(* IEC 61131-3 sources: std_i2980_v2.06_cp053/Source/IMM/ieccontrol/HostCommunication, 9 files *)

(* ---- ABDataSet.pu ---- *)
IMPORT_OVER_LISTFILE
 GET_SYNC_REFTO
, ASSERT
, STOP_PROCESS_ALGORITHM
, cDataSetErr_NoAvailable
, cDataSetErr_NotAllowed
, cModeAutomatic
, cCompOperationMode
, tevLockUnlock
, tsHostHmi
, tsHostDataSet
, tnDataState
, tnOperationMode
, KSYS_Status
, FBLockUnlock

END_IMPORT

ALGORITHM_BLOCK ABDataSet #DUMMY_EDIT_BLOCK

SYSTEM_VAR
 sv_bInitDone : BOOL (* IEC initialisation is finished (after movement registration) *);
 sv_HostHmi : tsHostHmi;
 sv_DataSet : tsHostDataSet;
 sv_DataState : tnDataState (* State of machine / mold data read *);
 sv_OperationMode : tnOperationMode;
END_VAR

SYSTEM_OBJECT
 TaskVis : TASK;
 evLockUnlock : tevLockUnlock;
 erAssert : ALARM;
END_OBJECT

VAR
 mpbAllowMoldLoad : REFTO BOOL;
 mpbAllowMoldSave : REFTO BOOL;
 mpbAllowMachineLoad : REFTO BOOL;
 mpbAllowMachineSave : REFTO BOOL;
 mpbAllowSeqLoad : REFTO BOOL;
 mpbAllowSeqSave : REFTO BOOL;
 mbOpModeLockAvailable : BOOL;
 mDataActionsEnableAvailable : BOOL;
END_VAR

FUNCTION fIsOpModeAutoAllowed : BOOL
 #DUMMY_EDIT_BLOCK
#BEGIN_EDIT_BLOCK

fIsOpModeAutoAllowed := NOT (sv_DataSet.iCommand = cDataSetCmdLoadMold) OR (sv_DataSet.iCommand = cDataSetCmdLoadMachine);

;#END_EDIT_BLOCK END_FUNCTION

FUNCTION fCheckConditions : BOOL
 #DUMMY_EDIT_BLOCK
#BEGIN_EDIT_BLOCK
IF (sv_DataState <> nReady) THEN
    RETURN;
END_IF;

IF (NOT fIsOpModeAutoAllowed()) THEN
    IF (sv_OperationMode >= nHalfAutomatic) THEN
        RETURN;
    END_IF;
END_IF;

fCheckConditions := TRUE;

;#END_EDIT_BLOCK END_FUNCTION

FUNCTION fDisableAll : BOOL
 #DUMMY_EDIT_BLOCK

VAR_INPUT
 bDisable : BOOL;
END_VAR
#BEGIN_EDIT_BLOCK
IF (mDataActionsEnableAvailable) THEN
   mpbAllowMoldLoad^ := NOT bDisable;
   mpbAllowMoldSave^ := NOT bDisable;
   mpbAllowMachineLoad^ := NOT bDisable;
   mpbAllowMachineSave^ := NOT bDisable;
   mpbAllowSeqLoad^ := NOT bDisable;
   mpbAllowSeqSave^ := NOT bDisable;
END_IF;

;#END_EDIT_BLOCK END_FUNCTION

POSTUPDATE_ALGORITHM pInit ON TaskVis(1) WITH sv_HostHmi.dataSet.bAvailable

VAR
 b : BOOL;
 s : KSYS_Status;
 dummy : DINT;
 dummyRef : REFTO UDINT;
END_VAR
#BEGIN_EDIT_BLOCK
mDataActionsEnableAvailable := TRUE;
mpbAllowMoldLoad := GET_SYNC_REFTO("system.sv_DataActionsEnable.bMoldDataLoad", T#0s, s);
mDataActionsEnableAvailable := mDataActionsEnableAvailable AND (s = KSYS_Status_OK);
mpbAllowMoldSave := GET_SYNC_REFTO("system.sv_DataActionsEnable.bMoldDataSave", T#0s, s);
mDataActionsEnableAvailable := mDataActionsEnableAvailable AND (s = KSYS_Status_OK);
mpbAllowMachineLoad := GET_SYNC_REFTO("system.sv_DataActionsEnable.bMachineDataLoad", T#0s, s);
mDataActionsEnableAvailable := mDataActionsEnableAvailable AND (s = KSYS_Status_OK);
mpbAllowMachineSave := GET_SYNC_REFTO("system.sv_DataActionsEnable.bMachineDataSave", T#0s, s);
mDataActionsEnableAvailable := mDataActionsEnableAvailable AND (s = KSYS_Status_OK);
mpbAllowSeqLoad := GET_SYNC_REFTO("system.sv_DataActionsEnable.bSequenceDataLoad", T#0s, s);
mDataActionsEnableAvailable := mDataActionsEnableAvailable AND (s = KSYS_Status_OK);
mpbAllowSeqSave := GET_SYNC_REFTO("system.sv_DataActionsEnable.bSequenceDataSave", T#0s, s);
mDataActionsEnableAvailable := mDataActionsEnableAvailable AND (s = KSYS_Status_OK);

dummyRef := GET_SYNC_REFTO("system.sv_LockOperationModeAuto.sResourceLock.iLocked", T#0s, s);
mbOpModeLockAvailable := s = KSYS_Status_OK;

IF (evLockUnlock = EMPTY) THEN
   dummy := Print("HostCommunication.ABDataSet: binary incompatible! recompile FU with correct iecproject!");
   b := ASSERT(FALSE, erAssert);
END_IF;

;#END_EDIT_BLOCK END_ALGORITHM

POSTUPDATE_ALGORITHM pTrigger ON TaskVis(2) WITH sv_DataSet.iTrigger

VAR
 b : BOOL;
END_VAR
#BEGIN_EDIT_BLOCK
IF (sv_DataSet.iTrigger MOD 2 = 0) THEN
    RETURN;
END_IF;

sv_DataSet.iError := 0;
IF (NOT sv_bInitDone) THEN
    sv_DataSet.iError := cDataSetErr_NotAllowed;
ELSIF (NOT sv_HostHmi.dataSet.bAvailable) THEN
    sv_DataSet.iError := cDataSetErr_NoAvailable;
ELSIF ((sv_DataSet.iCommand < cDataSetCmdLoadMold) OR (sv_DataSet.iCommand > cDataSetCmdSaveMachine)) THEN
    sv_DataSet.iError := cDataSetErr_InvalidCommand;
ELSIF (NOT fCheckConditions()) THEN
    sv_DataSet.iError := cDataSetErr_NotAllowed;
END_IF;

IF (sv_DataSet.iError > 0) THEN
    sv_DataSet.iTrigger := sv_DataSet.iTrigger + 1;
    RETURN;
END_IF;

b := fDisableAll(TRUE);

START_PROCESS_ALGORITHM(paRun);

;#END_EDIT_BLOCK END_ALGORITHM

PROCESS_ALGORITHM paRun ON TaskVis

VAR
 iStep : DINT;
 cnt : DINT;
 fbLockUnlock : FBLockUnlock;
 b : BOOL;
END_VAR
#BEGIN_EDIT_BLOCK
IF (iStep = 0) THEN
    IF (mbOpModeLockAvailable) THEN
        // op-mode will be locked by HMI (CR_0074160)
        iStep := 20;
    ELSE
        IF (NOT fIsOpModeAutoAllowed()) THEN
           fbLockUnlock.DeviceId.CompId := cCompOperationMode;
           fbLockUnlock.DeviceId.IndexId := 1;
           fbLockUnlock.MoveDir := cModeAutomatic;
           fbLockUnlock.MoveId := cModeAutomatic;
           fbLockUnlock(Mode := nLockAbort);
        END_IF;
        cnt := 10;
        iStep := 10;
    END_IF;
END_IF;

// CR_0074160: actually it is not possible to ensure there is no other load- or save-action in progress
// as a workaround lock the recipemask buttons and wait a second, then check conditions again
IF (iStep = 10) THEN
    cnt := cnt - 1;
    IF (cnt = 0) THEN
        iStep := 20;
    END_IF;
END_IF;

IF (iStep = 20) THEN
    IF (NOT fCheckConditions()) THEN
        sv_DataSet.iError := cDataSetErr_NotAllowed;
        iStep := 1000;
    ELSE
        iStep := 30;
    END_IF;
END_IF;

IF (iStep = 30) THEN
    sv_HostHmi.dataSet.iCommand := sv_DataSet.iCommand;
    sv_HostHmi.dataSet.sFile := sv_DataSet.sFile;
    sv_HostHmi.dataSet.iTrigger := sv_HostHmi.dataSet.iTrigger + 1;
    iStep := 40;
END_IF;

IF (iStep = 40) THEN
    IF (sv_HostHmi.dataSet.iTrigger MOD 2 = 0) THEN
        sv_DataSet.iError := sv_HostHmi.dataSet.iError;
        iStep := 1000;
    END_IF;
END_IF;

IF (iStep = 1000) THEN
    b := fDisableAll(FALSE);
    IF (NOT mbOpModeLockAvailable) THEN
        fbLockUnlock(Mode := nUnlock);
    END_IF;
    sv_DataSet.iTrigger := sv_DataSet.iTrigger + 1;
    iStep := 0;
    STOP_PROCESS_ALGORITHM();
END_IF;

;#END_EDIT_BLOCK END_ALGORITHM

END_ALGORITHM_BLOCK

#END_OF_IEC_PART

@Puma @IecEditor 6 159 @Pou 25
@@@BEG_Comment@@@

@@@END_Comment@@@

@BEG_Contents

@BEG_Func
@RT(17)FuncTreeContainer
3
@Var @RT(14)GET_SYNC_REFTO @RT(0) @T @T @DERIVED 0 @F @RT(22)KEBA_STANDARD_FUNCTION @F
@T
@BEG_Attrib
0 @RT(0) @RT(0)
@END_Attrib
1 1 @F @F @F @F

@Var @RT(6)ASSERT @RT(0) @T @T @DERIVED 0 @F @RT(8)FUNCTION @F
@T
@BEG_Attrib
0 @RT(0) @RT(0)
@END_Attrib
1 1 @F @F @F @F

@Var @RT(22)STOP_PROCESS_ALGORITHM @RT(0) @T @T @DERIVED 0 @F @RT(23)KEBA_STANDARD_PROCEDURE @F
@T
@BEG_Attrib
0 @RT(0) @RT(0)
@END_Attrib
1 1 @F @F @F @F

@END_Func

@BEG_Const
@RT(18)ConstTreeContainer
4
@Var @RT(23)cDataSetErr_NoAvailable @RT(0) @T @F @DT @RT(4)DINT @RT(0) @T @T @BASIC 0 @F
@F @F
@T
@BEG_Attrib
0 @RT(1)1 @RT(0)
@END_Attrib
1 1 @F @F @F @F

@Var @RT(22)cDataSetErr_NotAllowed @RT(0) @T @F @DT @RT(4)DINT @RT(0) @T @T @BASIC 0 @F
@F @F
@T
@BEG_Attrib
0 @RT(1)3 @RT(0)
@END_Attrib
1 1 @F @F @F @F

@Var @RT(14)cModeAutomatic @RT(0) @T @F @DT @RT(4)DINT @RT(0) @T @T @BASIC 0 @F
@F @F
@T
@BEG_Attrib
0 @RT(2)23 @RT(50)for locking/unlocking half and full automatic mode
@END_Attrib
1 1 @F @F @F @F

@Var @RT(18)cCompOperationMode @RT(0) @T @F @DT @RT(4)DINT @RT(0) @T @T @BASIC 0 @F
@F @F
@T
@BEG_Attrib
0 @RT(3)111 @RT(24)Component Operation Mode
@END_Attrib
1 1 @F @F @F @F

@END_Const

@BEG_Export

@BEG_Kind
@ALGORITHM_BLOCK @RT(9)ABDataSet @STRUCTURED_TEXT
@RT(0) @RT(0) @RT(0)
@END_Kind

@BEG_Dcl
@RT(16)DclTreeContainer
16
@Var @RT(7)TaskVis @RT(0) @T @T @RENAMED 0 @T @T @DT @RT(4)TASK @RT(0) @T @T @BASIC 0 @F
@F @F
@T
@BEG_Attrib
3 @RT(0) @RT(0) @RT(0)
@END_Attrib
1 7 @F @F @F @F

@Var @RT(12)sv_bInitDone @RT(0) @T @F @DT @RT(4)BOOL @RT(0) @T @T @BASIC 0 @F
@F @F
@T
@BEG_Attrib
3 @RT(0) @RT(60)IEC initialisation is finished (after movement registration) @RT(0)
@END_Attrib
1 8 @F @F @F @F

@Var @RT(12)evLockUnlock @RT(0) @T @T @DERIVED 0 @T @T @DT @RT(13)tevLockUnlock @RT(0) @T @T @UNKNOWN 0 @F
@F @F
@T
@BEG_Attrib
3 @RT(0) @RT(0) @RT(0)
@END_Attrib
1 7 @F @F @F @F

@Var @RT(10)sv_HostHmi @RT(0) @T @T @DERIVED 0 @T @T @DT @RT(9)tsHostHmi @RT(0) @T @T @UNKNOWN 0 @F
@F @F
@T
@BEG_Attrib
3 @RT(0) @RT(0) @RT(0)
@END_Attrib
1 8 @F @F @F @F

@Var @RT(10)sv_DataSet @RT(0) @T @T @DERIVED 0 @T @T @DT @RT(13)tsHostDataSet @RT(0) @T @T @UNKNOWN 0 @F
@F @F
@T
@BEG_Attrib
3 @RT(0) @RT(0) @RT(0)
@END_Attrib
1 8 @F @F @F @F

@Var @RT(12)sv_DataState @RT(0) @T @T @DERIVED 0 @T @T @DT @RT(11)tnDataState @RT(0) @T @T @UNKNOWN 0 @F
@F @F
@T
@BEG_Attrib
3 @RT(0) @RT(33)State of machine / mold data read @RT(0)
@END_Attrib
1 8 @F @F @F @F

@Var @RT(16)sv_OperationMode @RT(0) @T @T @DERIVED 0 @T @T @DT @RT(15)tnOperationMode @RT(0) @T @T @UNKNOWN 0 @F
@F @F
@T
@BEG_Attrib
3 @RT(0) @RT(0) @RT(0)
@END_Attrib
1 8 @F @F @F @F

@Var @RT(8)erAssert @RT(0) @T @F @DT @RT(5)ALARM @RT(0) @T @T @BASIC 0 @F
@F @F
@T
@BEG_Attrib
3 @RT(0) @RT(0) @RT(0)
@END_Attrib
1 7 @F @F @F @F

@Var @RT(16)mpbAllowMoldLoad @RT(0) @T @T @REFTO 0 @T @DT @RT(4)BOOL @RT(0) @T @T @BASIC 0 @F
@F @F
@T
@BEG_Attrib
3 @RT(0) @RT(0) @RT(0)
@END_Attrib
1 0 @F @F @F @F

@Var @RT(16)mpbAllowMoldSave @RT(0) @T @T @REFTO 0 @T @DT @RT(4)BOOL @RT(0) @T @T @BASIC 0 @F
@F @F
@T
@BEG_Attrib
3 @RT(0) @RT(0) @RT(0)
@END_Attrib
1 0 @F @F @F @F

@Var @RT(19)mpbAllowMachineLoad @RT(0) @T @T @REFTO 0 @T @DT @RT(4)BOOL @RT(0) @T @T @BASIC 0 @F
@F @F
@T
@BEG_Attrib
3 @RT(0) @RT(0) @RT(0)
@END_Attrib
1 0 @F @F @F @F

@Var @RT(19)mpbAllowMachineSave @RT(0) @T @T @REFTO 0 @T @DT @RT(4)BOOL @RT(0) @T @T @BASIC 0 @F
@F @F
@T
@BEG_Attrib
3 @RT(0) @RT(0) @RT(0)
@END_Attrib
1 0 @F @F @F @F

@Var @RT(15)mpbAllowSeqLoad @RT(0) @T @T @REFTO 0 @T @DT @RT(4)BOOL @RT(0) @T @T @BASIC 0 @F
@F @F
@T
@BEG_Attrib
3 @RT(0) @RT(0) @RT(0)
@END_Attrib
1 0 @F @F @F @F

@Var @RT(15)mpbAllowSeqSave @RT(0) @T @T @REFTO 0 @T @DT @RT(4)BOOL @RT(0) @T @T @BASIC 0 @F
@F @F
@T
@BEG_Attrib
3 @RT(0) @RT(0) @RT(0)
@END_Attrib
1 0 @F @F @F @F

@Var @RT(21)mbOpModeLockAvailable @RT(0) @T @F @DT @RT(4)BOOL @RT(0) @T @T @BASIC 0 @F
@F @F
@T
@BEG_Attrib
3 @RT(0) @RT(0) @RT(0)
@END_Attrib
1 0 @F @F @F @F

@Var @RT(27)mDataActionsEnableAvailable @RT(0) @T @F @DT @RT(4)BOOL @RT(0) @T @T @BASIC 0 @F
@F @F
@T
@BEG_Attrib
3 @RT(0) @RT(0) @RT(0)
@END_Attrib
1 0 @F @F @F @F

@END_Dcl

@END_Export

@BEG_Body

6

@BEG_Export

@BEG_Algo
@FUNCTION @RT(20)fIsOpModeAutoAllowed @STRUCTURED_TEXT
@RT(4)BOOL @RT(0) @RT(0) @F @F
@END_Algo

@BEG_Dcl
@RT(16)DclTreeContainer
0
@END_Dcl

@END_Export

@BEG_Export

@BEG_Algo
@FUNCTION @RT(16)fCheckConditions @STRUCTURED_TEXT
@RT(4)BOOL @RT(0) @RT(0) @F @F
@END_Algo

@BEG_Dcl
@RT(16)DclTreeContainer
0
@END_Dcl

@END_Export

@BEG_Export

@BEG_Algo
@FUNCTION @RT(11)fDisableAll @STRUCTURED_TEXT
@RT(4)BOOL @RT(0) @RT(0) @F @F
@END_Algo

@BEG_Dcl
@RT(16)DclTreeContainer
1
@Var @RT(8)bDisable @RT(0) @T @F @DT @RT(4)BOOL @RT(0) @T @T @BASIC 0 @F
@F @F
@T
@BEG_Attrib
3 @RT(0) @RT(0) @RT(0)
@END_Attrib
1 1 @F @F @F @F

@END_Dcl

@END_Export

@BEG_Export

@BEG_Algo
@POSTUPDATE_ALGORITHM @RT(5)pInit @STRUCTURED_TEXT
@RT(0) @RT(29)sv_HostHmi.dataSet.bAvailable @RT(10)TaskVis(1) @F @F
@END_Algo

@BEG_Dcl
@RT(16)DclTreeContainer
4
@Var @RT(1)b @RT(0) @T @F @DT @RT(4)BOOL @RT(0) @T @T @BASIC 0 @F
@F @F
@T
@BEG_Attrib
3 @RT(0) @RT(0) @RT(0)
@END_Attrib
1 0 @F @F @F @F

@Var @RT(1)s @RT(0) @T @T @DERIVED 0 @T @T @DT @RT(11)KSYS_Status @RT(0) @T @T @UNKNOWN 0 @F
@F @F
@T
@BEG_Attrib
3 @RT(0) @RT(0) @RT(0)
@END_Attrib
1 0 @F @F @F @F

@Var @RT(5)dummy @RT(0) @T @F @DT @RT(4)DINT @RT(0) @T @T @BASIC 0 @F
@F @F
@T
@BEG_Attrib
3 @RT(0) @RT(0) @RT(0)
@END_Attrib
1 0 @F @F @F @F

@Var @RT(8)dummyRef @RT(0) @T @T @REFTO 0 @T @DT @RT(5)UDINT @RT(0) @T @T @BASIC 0 @F
@F @F
@T
@BEG_Attrib
3 @RT(0) @RT(0) @RT(0)
@END_Attrib
1 0 @F @F @F @F

@END_Dcl

@END_Export

@BEG_Export

@BEG_Algo
@POSTUPDATE_ALGORITHM @RT(8)pTrigger @STRUCTURED_TEXT
@RT(0) @RT(19)sv_DataSet.iTrigger @RT(10)TaskVis(2) @F @F
@END_Algo

@BEG_Dcl
@RT(16)DclTreeContainer
1
@Var @RT(1)b @RT(0) @T @F @DT @RT(4)BOOL @RT(0) @T @T @BASIC 0 @F
@F @F
@T
@BEG_Attrib
3 @RT(0) @RT(0) @RT(0)
@END_Attrib
1 0 @F @F @F @F

@END_Dcl

@END_Export

@BEG_Export

@BEG_Algo
@PROCESS_ALGORITHM @RT(5)paRun @STRUCTURED_TEXT
@RT(0) @RT(0) @RT(7)TaskVis @F @F
@END_Algo

@BEG_Dcl
@RT(16)DclTreeContainer
4
@Var @RT(5)iStep @RT(0) @T @F @DT @RT(4)DINT @RT(0) @T @T @BASIC 0 @F
@F @F
@T
@BEG_Attrib
3 @RT(0) @RT(0) @RT(0)
@END_Attrib
1 0 @F @F @F @F

@Var @RT(3)cnt @RT(0) @T @F @DT @RT(4)DINT @RT(0) @T @T @BASIC 0 @F
@F @F
@T
@BEG_Attrib
3 @RT(0) @RT(0) @RT(0)
@END_Attrib
1 0 @F @F @F @F

@Var @RT(12)fbLockUnlock @RT(0) @T @T @DERIVED 0 @T @T @DT @RT(12)FBLockUnlock @RT(0) @T @T @UNKNOWN 0 @F
@F @F
@T
@BEG_Attrib
3 @RT(0) @RT(0) @RT(0)
@END_Attrib
1 0 @F @F @F @F

@Var @RT(1)b @RT(0) @T @F @DT @RT(4)BOOL @RT(0) @T @T @BASIC 0 @F
@F @F
@T
@BEG_Attrib
3 @RT(0) @RT(0) @RT(0)
@END_Attrib
1 0 @F @F @F @F

@END_Dcl

@END_Export

@BEG_Body
@TL(3)

fIsOpModeAutoAllowed := NOT (sv_DataSet.iCommand = cDataSetCmdLoadMold) OR (sv_DataSet.iCommand = cDataSetCmdLoadMachine);

@END_Body

@@@BEG_Comment@@@
@TL(0)

@@@END_Comment@@@

@BEG_Body
@TL(12)
IF (sv_DataState <> nReady) THEN
    RETURN;
END_IF;

IF (NOT fIsOpModeAutoAllowed()) THEN
    IF (sv_OperationMode >= nHalfAutomatic) THEN
        RETURN;
    END_IF;
END_IF;

fCheckConditions := TRUE;

@END_Body

@@@BEG_Comment@@@
@TL(0)

@@@END_Comment@@@

@BEG_Body
@TL(9)
IF (mDataActionsEnableAvailable) THEN
   mpbAllowMoldLoad^ := NOT bDisable;
   mpbAllowMoldSave^ := NOT bDisable;
   mpbAllowMachineLoad^ := NOT bDisable;
   mpbAllowMachineSave^ := NOT bDisable;
   mpbAllowSeqLoad^ := NOT bDisable;
   mpbAllowSeqSave^ := NOT bDisable;
END_IF;

@END_Body

@@@BEG_Comment@@@
@TL(0)

@@@END_Comment@@@

@BEG_Body
@TL(22)
mDataActionsEnableAvailable := TRUE;
mpbAllowMoldLoad := GET_SYNC_REFTO("system.sv_DataActionsEnable.bMoldDataLoad", T#0s, s);
mDataActionsEnableAvailable := mDataActionsEnableAvailable AND (s = KSYS_Status_OK);
mpbAllowMoldSave := GET_SYNC_REFTO("system.sv_DataActionsEnable.bMoldDataSave", T#0s, s);
mDataActionsEnableAvailable := mDataActionsEnableAvailable AND (s = KSYS_Status_OK);
mpbAllowMachineLoad := GET_SYNC_REFTO("system.sv_DataActionsEnable.bMachineDataLoad", T#0s, s);
mDataActionsEnableAvailable := mDataActionsEnableAvailable AND (s = KSYS_Status_OK);
mpbAllowMachineSave := GET_SYNC_REFTO("system.sv_DataActionsEnable.bMachineDataSave", T#0s, s);
mDataActionsEnableAvailable := mDataActionsEnableAvailable AND (s = KSYS_Status_OK);
mpbAllowSeqLoad := GET_SYNC_REFTO("system.sv_DataActionsEnable.bSequenceDataLoad", T#0s, s);
mDataActionsEnableAvailable := mDataActionsEnableAvailable AND (s = KSYS_Status_OK);
mpbAllowSeqSave := GET_SYNC_REFTO("system.sv_DataActionsEnable.bSequenceDataSave", T#0s, s);
mDataActionsEnableAvailable := mDataActionsEnableAvailable AND (s = KSYS_Status_OK);

dummyRef := GET_SYNC_REFTO("system.sv_LockOperationModeAuto.sResourceLock.iLocked", T#0s, s);
mbOpModeLockAvailable := s = KSYS_Status_OK;

IF (evLockUnlock = EMPTY) THEN
   dummy := Print("HostCommunication.ABDataSet: binary incompatible! recompile FU with correct iecproject!");
   b := ASSERT(FALSE, erAssert);
END_IF;

@END_Body

@@@BEG_Comment@@@
@TL(0)

@@@END_Comment@@@

@BEG_Body
@TL(24)
IF (sv_DataSet.iTrigger MOD 2 = 0) THEN
    RETURN;
END_IF;

sv_DataSet.iError := 0;
IF (NOT sv_bInitDone) THEN
    sv_DataSet.iError := cDataSetErr_NotAllowed;
ELSIF (NOT sv_HostHmi.dataSet.bAvailable) THEN
    sv_DataSet.iError := cDataSetErr_NoAvailable;
ELSIF ((sv_DataSet.iCommand < cDataSetCmdLoadMold) OR (sv_DataSet.iCommand > cDataSetCmdSaveMachine)) THEN
    sv_DataSet.iError := cDataSetErr_InvalidCommand;
ELSIF (NOT fCheckConditions()) THEN
    sv_DataSet.iError := cDataSetErr_NotAllowed;
END_IF;

IF (sv_DataSet.iError > 0) THEN
    sv_DataSet.iTrigger := sv_DataSet.iTrigger + 1;
    RETURN;
END_IF;

b := fDisableAll(TRUE);

START_PROCESS_ALGORITHM(paRun);

@END_Body

@@@BEG_Comment@@@
@TL(0)

@@@END_Comment@@@

@BEG_Body
@TL(61)
IF (iStep = 0) THEN
    IF (mbOpModeLockAvailable) THEN
        // op-mode will be locked by HMI (CR_0074160)
        iStep := 20;
    ELSE
        IF (NOT fIsOpModeAutoAllowed()) THEN
           fbLockUnlock.DeviceId.CompId := cCompOperationMode;
           fbLockUnlock.DeviceId.IndexId := 1;
           fbLockUnlock.MoveDir := cModeAutomatic;
           fbLockUnlock.MoveId := cModeAutomatic;
           fbLockUnlock(Mode := nLockAbort);
        END_IF;
        cnt := 10;
        iStep := 10;
    END_IF;
END_IF;

// CR_0074160: actually it is not possible to ensure there is no other load- or save-action in progress
// as a workaround lock the recipemask buttons and wait a second, then check conditions again
IF (iStep = 10) THEN
    cnt := cnt - 1;
    IF (cnt = 0) THEN
        iStep := 20;
    END_IF;
END_IF;

IF (iStep = 20) THEN
    IF (NOT fCheckConditions()) THEN
        sv_DataSet.iError := cDataSetErr_NotAllowed;
        iStep := 1000;
    ELSE
        iStep := 30;
    END_IF;
END_IF;

IF (iStep = 30) THEN
    sv_HostHmi.dataSet.iCommand := sv_DataSet.iCommand;
    sv_HostHmi.dataSet.sFile := sv_DataSet.sFile;
    sv_HostHmi.dataSet.iTrigger := sv_HostHmi.dataSet.iTrigger + 1;
    iStep := 40;
END_IF;

IF (iStep = 40) THEN
    IF (sv_HostHmi.dataSet.iTrigger MOD 2 = 0) THEN
        sv_DataSet.iError := sv_HostHmi.dataSet.iError;
        iStep := 1000;
    END_IF;
END_IF;

IF (iStep = 1000) THEN
    b := fDisableAll(FALSE);
    IF (NOT mbOpModeLockAvailable) THEN
        fbLockUnlock(Mode := nUnlock);
    END_IF;
    sv_DataSet.iTrigger := sv_DataSet.iTrigger + 1;
    iStep := 0;
    STOP_PROCESS_ALGORITHM();
END_IF;

@END_Body

@@@BEG_Comment@@@
@TL(0)

@@@END_Comment@@@
@END_Body

@END_Contents

(* ---- ABHeatingState.pu ---- *)
(*
Euromap63 and 83 specific heating zone states
*)

IMPORT_OVER_LISTFILE
 tsEM77
, tsEM63
, tenEM83ZoneMode
, tsHeatingGeneral
, tsHeatingZone
, KSYS_Status
, tyHeatingNozzle
, tyHeatingMold
, RTC
, tyHeatingNozzleGeneral

END_IMPORT

ALGORITHM_BLOCK ABHeatingState #DUMMY_EDIT_BLOCK

SYSTEM_VAR
 sv_EM77 : tsEM77;
 sv_EM63 : tsEM63;
END_VAR

VAR
 mbEM63 : BOOL;
END_VAR

FUNCTION fZoneModeToString : STRING(1)
 #DUMMY_EDIT_BLOCK

VAR_INPUT
 zoneMode : tenEM83ZoneMode;
END_VAR
#BEGIN_EDIT_BLOCK
(**************************************** WARNING ********************************************
 *** The KEBA Kemro K2 System including software is not intended for safety control tasks! ***
 ***                       For further information see Comment tab!                        ***
 *********************************************************************************************)

// mapping from EM83 zone mode (14.6 Table 63) to EM63 zone mode

//    "0" Barrel Zone is not supported    ... EM83: OTHER_0
//    "O" Barrel Zone is off              ... EM83: OFF_1, ONLY_MEASUREMENT_6
//    "A" Barrel Zone is in auto mode     ... EM83: AUTOMATIC_2
//    "T" Barrel Zone is in tuning mode   ... EM83: TUNING_3
//    "S" Barrel Zone is in standby mode  ... EM83: STANDBY_4
//    "M" Barrel Zone is in manual mode   ... EM83: OPEN_LOOP_5

CASE (zoneMode) OF
    nOther_0: fZoneModeToString := "0";
    nOff_1: fZoneModeToString := "O";
    nOnlyMeasurement_6: fZoneModeToString := "O";
    nAutomatic_2: fZoneModeToString := "A";
    nTuning_3: fZoneModeToString := "T";
    nStandby_4: fZoneModeToString := "S";
    nOpenLoop_5: fZoneModeToString := "M";

ELSE
    fZoneModeToString := "0";
END_CASE;

;#END_EDIT_BLOCK END_FUNCTION

FUNCTION fUpdateHeatingZone : BOOL
 #DUMMY_EDIT_BLOCK

VAR_INPUT
 iZoneNr : DINT;
END_VAR

VAR_IN_OUT
 general : tsHeatingGeneral;
 zone : tsHeatingZone;
 zoneModeEM63 : STRING(1);
 zoneModeEM83 : tenEM83ZoneMode;
END_VAR

VAR
 zoneMode : tenEM83ZoneMode;
END_VAR
#BEGIN_EDIT_BLOCK
(**************************************** WARNING ********************************************
 *** The KEBA Kemro K2 System including software is not intended for safety control tasks! ***
 ***                       For further information see Comment tab!                        ***
 *********************************************************************************************)

IF (zone.pZoneMode = EMPTY) THEN
   RETURN;
END_IF;

IF (general.piZonesAvailable <> EMPTY) AND (iZoneNr > general.piZonesAvailable^) THEN
    zoneMode := nOther_0;
ELSIF (general.pbHeatingOn <> EMPTY) AND (NOT general.pbHeatingOn^) THEN
    zoneMode := nOff_1;
ELSIF NOT (zone.pbUsed^) THEN
    zoneMode := nOff_1;
ELSIF (zone.pZoneMode^ = enZoneModeDisabled)  THEN
    zoneMode := nOff_1;
ELSIF (zone.pZoneMode^ = enZoneModeMeasure) THEN
    zoneMode := nOnlyMeasurement_6;
ELSIF (zone.pZoneMode^ = enZoneModeConstant) THEN
    zoneMode := nOpenLoop_5;
ELSIF (zone.pbOptimizingActive^) THEN
    zoneMode := nTuning_3;
ELSIF ((general.pbKeepWarmActive <> EMPTY) AND (general.pbKeepWarmActive^)) THEN
    zoneMode := nStandby_4;
ELSE
    zoneMode := nAutomatic_2;
END_IF;

IF (zoneModeEM83 <> zoneMode) THEN
    zoneModeEM83 := zoneMode;
    IF (mbEM63) THEN
       zoneModeEM63 := fZoneModeToString(zoneMode);
    END_IF;
END_IF;

fUpdateHeatingZone := TRUE;

;#END_EDIT_BLOCK END_FUNCTION

FUNCTION fInitHeatingZone : BOOL
 #DUMMY_EDIT_BLOCK

VAR_INPUT
 sPrefix : STRING(31);
 iZoneNr : DINT;
END_VAR

VAR_IN_OUT
 zone : tsHeatingZone;
END_VAR

VAR
 sPrefixZone : STRING(127);
 s : KSYS_Status;
 pbLinked : REFTO BOOL;
END_VAR
#BEGIN_EDIT_BLOCK
(**************************************** WARNING ********************************************
 *** The KEBA Kemro K2 System including software is not intended for safety control tasks! ***
 ***                       For further information see Comment tab!                        ***
 *********************************************************************************************)

pbLinked := GET_SYNC_REFTO(CONCAT(sPrefix, "Array[", DINT_TO_STRING(iZoneNr),"].bLinked"), T#0s, s);
IF ((pbLinked =EMPTY) OR (NOT pbLinked^)) THEN
    RETURN;
END_IF;

sPrefixZone := CONCAT(sPrefix, DINT_TO_STRING(iZoneNr));
zone.pbOptimizingActive := GET_SYNC_REFTO(CONCAT(sPrefixZone, ".bIsOptimizing"), t#0s, s);
zone.pbEmergencyOperation := GET_SYNC_REFTO(CONCAT(sPrefixZone, ".bEmgOperation"), t#0s, s);

sPrefixZone := CONCAT(sPrefix, "Retain", DINT_TO_STRING(iZoneNr));
zone.pZoneMode := GET_SYNC_REFTO(CONCAT(sPrefixZone, ".ModeVis"), t#0s, s);
zone.pbUsed := GET_SYNC_REFTO(CONCAT(sPrefixZone, ".bUsed"), t#0s, s);

fInitHeatingZone := TRUE;

;#END_EDIT_BLOCK END_FUNCTION

ALGORITHM aHeating

VAR_INPUT
 bEM63 : BOOL;
END_VAR

VAR_TEMP
 k : DINT;
 i : DINT;
END_VAR

VAR
 yHeatingZonesNozzle : tyHeatingNozzle;
 yHeatingZonesMold : tyHeatingMold;
 bInit : BOOL;
 rtc : RTC;
 ts : DT;
 t : TIME;
 b : BOOL;
 sPrefix : STRING(63);
 mHeatingMoldGeneral : tsHeatingGeneral;
 mHeatingNozzleGeneral : tyHeatingNozzleGeneral;
 s : KSYS_Status;
END_VAR
#BEGIN_EDIT_BLOCK
(**************************************** WARNING ********************************************
 *** The KEBA Kemro K2 System including software is not intended for safety control tasks! ***
 ***                       For further information see Comment tab!                        ***
 *********************************************************************************************)

// SetCfgBrlZn, SetCfgMldZn

IF (NOT bInit) THEN
    mbEM63 := bEM63;
    rtc();
    ts := rtc.CDT;
    bInit := TRUE;
    FOR k := 1 TO cMaxInjectionUnits DO
        sPrefix := CONCAT("HeatingNozzle", DINT_TO_STRING(k));
        mHeatingNozzleGeneral[k].pbKeepWarmActive := GET_SYNC_REFTO(CONCAT(sPrefix, ".sv_bKeepWarmActive"), T#0s, s);
        mHeatingNozzleGeneral[k].pbHeatingOn := GET_SYNC_REFTO(CONCAT(sPrefix, ".sv_bHeatingOn"), T#0s, s);
        mHeatingNozzleGeneral[k].piZonesAvailable := GET_SYNC_REFTO(CONCAT(sPrefix, ".sv_iZonesAvailable"), T#0s, s);
        sPrefix := CONCAT(sPrefix, ".sv_Zone");

        FOR i := 1 TO cMaxHeatingNozzleZones DO
            b := fInitHeatingZone(sPrefix, i, yHeatingZonesNozzle[k, i]);
            IF (NOT b) THEN
               EXIT;
            END_IF;
        END_FOR;
    END_FOR;

    sPrefix := "HeatingMold1.sv_Zone";
    mHeatingMoldGeneral.pbKeepWarmActive := GET_SYNC_REFTO("HeatingMold1.sv_bKeepWarmActive", T#0s, s);
    mHeatingMoldGeneral.pbHeatingOn := GET_SYNC_REFTO("HeatingMold1.sv_bHeatingOn", T#0s, s);
    mHeatingMoldGeneral.piZonesAvailable := GET_SYNC_REFTO("HeatingMold1.sv_iZonesAvailable", T#0s, s);
    FOR i := 1 TO cMaxHeatingMoldZones DO
        b := fInitHeatingZone(sPrefix, i, yHeatingZonesMold[i]);
        IF (NOT b) THEN
            EXIT;
        END_IF;
    END_FOR;

    rtc();
    t := rtc.CDT - ts;

END_IF;

FOR k := 1 TO cMaxInjectionUnits DO
    FOR i := 1 TO cMaxHeatingNozzleZones DO
        b := fUpdateHeatingZone(i, mHeatingNozzleGeneral[k], yHeatingZonesNozzle[k,i], sv_EM63.SetCfgBrlZn[k,i], sv_EM77.SetCfgBrlZn[k,i]);
        IF (NOT b) THEN
           EXIT;
        END_IF;
    END_FOR;
END_FOR;

FOR i := 1 TO cMaxHeatingMoldZones DO
    b := fUpdateHeatingZone(i, mHeatingMoldGeneral, yHeatingZonesMold[i], sv_EM63.SetCfgMldZn[i], sv_EM77.SetCfgMldZn[i]);
    IF (NOT b) THEN
        EXIT;
    END_IF;
END_FOR;

;#END_EDIT_BLOCK END_ALGORITHM

END_ALGORITHM_BLOCK

#END_OF_IEC_PART

@Puma @IecEditor 6 168 @Pou 25
@@@BEG_Comment@@@
Euromap63 and 83 specific heating zone states
@@@END_Comment@@@

@BEG_Contents

@BEG_Func
@RT(17)FuncTreeContainer
0
@END_Func

@BEG_Const
@RT(18)ConstTreeContainer
0
@END_Const

@BEG_Export

@BEG_Kind
@ALGORITHM_BLOCK @RT(14)ABHeatingState @STRUCTURED_TEXT
@RT(0) @RT(0) @RT(0)
@END_Kind

@BEG_Dcl
@RT(16)DclTreeContainer
3
@Var @RT(7)sv_EM77 @RT(0) @T @T @DERIVED 0 @F @RT(6)tsEM77 @F
@T
@BEG_Attrib
3 @RT(0) @RT(0) @RT(0)
@END_Attrib
1 8 @F @F @F @F

@Var @RT(7)sv_EM63 @RT(0) @T @T @DERIVED 0 @F @RT(6)tsEM63 @F
@T
@BEG_Attrib
3 @RT(0) @RT(0) @RT(0)
@END_Attrib
1 8 @F @F @F @F

@Var @RT(6)mbEM63 @RT(0) @T @F @DT @RT(4)BOOL @RT(0) @T @T @BASIC 0 @F
@F @F
@T
@BEG_Attrib
3 @RT(0) @RT(0) @RT(0)
@END_Attrib
1 0 @F @F @F @F

@END_Dcl

@END_Export

@BEG_Body

4

@BEG_Export

@BEG_Algo
@FUNCTION @RT(17)fZoneModeToString @STRUCTURED_TEXT
@RT(9)STRING(1) @RT(0) @RT(0) @F @F
@END_Algo

@BEG_Dcl
@RT(16)DclTreeContainer
1
@Var @RT(8)zoneMode @RT(0) @T @T @DERIVED 0 @T @T @DT @RT(15)tenEM83ZoneMode @RT(0) @T @T @UNKNOWN 0 @F
@F @F
@T
@BEG_Attrib
3 @RT(0) @RT(0) @RT(0)
@END_Attrib
1 1 @F @F @F @F

@END_Dcl

@END_Export

@BEG_Export

@BEG_Algo
@FUNCTION @RT(18)fUpdateHeatingZone @STRUCTURED_TEXT
@RT(4)BOOL @RT(0) @RT(0) @F @F
@END_Algo

@BEG_Dcl
@RT(16)DclTreeContainer
6
@Var @RT(7)iZoneNr @RT(0) @T @F @DT @RT(4)DINT @RT(0) @T @T @BASIC 0 @F
@F @F
@T
@BEG_Attrib
3 @RT(0) @RT(0) @RT(0)
@END_Attrib
1 1 @F @F @F @F

@Var @RT(7)general @RT(0) @T @T @DERIVED 0 @T @T @DT @RT(16)tsHeatingGeneral @RT(0) @T @T @UNKNOWN 0 @F
@F @F
@T
@BEG_Attrib
3 @RT(0) @RT(0) @RT(0)
@END_Attrib
1 2 @F @F @F @F

@Var @RT(4)zone @RT(0) @T @T @DERIVED 0 @F @RT(13)tsHeatingZone @F
@T
@BEG_Attrib
3 @RT(0) @RT(0) @RT(0)
@END_Attrib
1 2 @F @F @F @F

@Var @RT(12)zoneModeEM63 @RT(0) @T @F @DT @RT(9)STRING(1) @RT(0) @T @T @STRING 0 @F @RT(1)1 @F
@F @F
@T
@BEG_Attrib
3 @RT(0) @RT(0) @RT(0)
@END_Attrib
1 2 @F @F @F @F

@Var @RT(8)zoneMode @RT(0) @T @T @DERIVED 0 @T @T @DT @RT(15)tenEM83ZoneMode @RT(0) @T @T @UNKNOWN 0 @F
@F @F
@T
@BEG_Attrib
3 @RT(0) @RT(0) @RT(0)
@END_Attrib
1 0 @F @F @F @F

@Var @RT(12)zoneModeEM83 @RT(0) @T @T @DERIVED 0 @F @RT(15)tenEM83ZoneMode @F
@T
@BEG_Attrib
3 @RT(0) @RT(0) @RT(0)
@END_Attrib
1 2 @F @F @F @F

@END_Dcl

@END_Export

@BEG_Export

@BEG_Algo
@FUNCTION @RT(16)fInitHeatingZone @STRUCTURED_TEXT
@RT(4)BOOL @RT(0) @RT(0) @F @F
@END_Algo

@BEG_Dcl
@RT(16)DclTreeContainer
6
@Var @RT(7)sPrefix @RT(0) @T @F @DT @RT(10)STRING(31) @RT(0) @T @T @STRING 0 @F @RT(2)31 @F
@F @F
@T
@BEG_Attrib
3 @RT(0) @RT(0) @RT(0)
@END_Attrib
1 1 @F @F @F @F

@Var @RT(7)iZoneNr @RT(0) @T @F @DT @RT(4)DINT @RT(0) @T @T @BASIC 0 @F
@F @F
@T
@BEG_Attrib
3 @RT(0) @RT(0) @RT(0)
@END_Attrib
1 1 @F @F @F @F

@Var @RT(4)zone @RT(0) @T @T @DERIVED 0 @T @T @DT @RT(13)tsHeatingZone @RT(0) @T @T @UNKNOWN 0 @F
@F @F
@T
@BEG_Attrib
3 @RT(0) @RT(0) @RT(0)
@END_Attrib
1 2 @F @F @F @F

@Var @RT(11)sPrefixZone @RT(0) @T @F @DT @RT(11)STRING(127) @RT(0) @T @T @STRING 0 @F @RT(3)127 @F
@F @F
@T
@BEG_Attrib
3 @RT(0) @RT(0) @RT(0)
@END_Attrib
1 0 @F @F @F @F

@Var @RT(1)s @RT(0) @T @T @DERIVED 0 @T @T @DT @RT(11)KSYS_Status @RT(0) @T @T @UNKNOWN 0 @F
@F @F
@T
@BEG_Attrib
3 @RT(0) @RT(0) @RT(0)
@END_Attrib
1 0 @F @F @F @F

@Var @RT(8)pbLinked @RT(0) @T @T @REFTO 0 @T @DT @RT(4)BOOL @RT(0) @T @T @BASIC 0 @F
@F @F
@T
@BEG_Attrib
3 @RT(0) @RT(0) @RT(0)
@END_Attrib
1 0 @F @F @F @F

@END_Dcl

@END_Export

@BEG_Export

@BEG_Algo
@ALGORITHM @RT(8)aHeating @STRUCTURED_TEXT
@RT(0) @RT(0) @RT(0) @F @F
@END_Algo

@BEG_Dcl
@RT(16)DclTreeContainer
14
@Var @RT(19)yHeatingZonesNozzle @RT(0) @T @T @DERIVED 0 @T @T @DT @RT(15)tyHeatingNozzle @RT(0) @T @T @UNKNOWN 0 @F
@F @F
@T
@BEG_Attrib
3 @RT(0) @RT(0) @RT(0)
@END_Attrib
1 0 @F @F @F @F

@Var @RT(17)yHeatingZonesMold @RT(0) @T @T @DERIVED 0 @T @T @DT @RT(13)tyHeatingMold @RT(0) @T @T @UNKNOWN 0 @F
@F @F
@T
@BEG_Attrib
3 @RT(0) @RT(0) @RT(0)
@END_Attrib
1 0 @F @F @F @F

@Var @RT(5)bInit @RT(0) @T @F @DT @RT(4)BOOL @RT(0) @T @T @BASIC 0 @F
@F @F
@T
@BEG_Attrib
3 @RT(0) @RT(0) @RT(0)
@END_Attrib
1 0 @F @F @F @F

@Var @RT(3)rtc @RT(0) @T @T @DERIVED 0 @T @T @DT @RT(3)RTC @RT(0) @T @T @UNKNOWN 0 @F
@F @F
@T
@BEG_Attrib
3 @RT(0) @RT(0) @RT(0)
@END_Attrib
1 0 @F @F @F @F

@Var @RT(2)ts @RT(0) @T @F @DT @RT(2)DT @RT(0) @T @T @BASIC 0 @F
@F @F
@T
@BEG_Attrib
3 @RT(0) @RT(0) @RT(0)
@END_Attrib
1 0 @F @F @F @F

@Var @RT(1)t @RT(0) @T @F @DT @RT(4)TIME @RT(0) @T @T @BASIC 0 @F
@F @F
@T
@BEG_Attrib
3 @RT(0) @RT(0) @RT(0)
@END_Attrib
1 0 @F @F @F @F

@Var @RT(1)b @RT(0) @T @F @DT @RT(4)BOOL @RT(0) @T @T @BASIC 0 @F
@F @F
@T
@BEG_Attrib
3 @RT(0) @RT(0) @RT(0)
@END_Attrib
1 0 @F @F @F @F

@Var @RT(1)k @RT(0) @T @F @DT @RT(4)DINT @RT(0) @T @T @BASIC 0 @F
@F @F
@T
@BEG_Attrib
3 @RT(0) @RT(0) @RT(0)
@END_Attrib
1 4 @F @F @F @F

@Var @RT(1)i @RT(0) @T @F @DT @RT(4)DINT @RT(0) @T @T @BASIC 0 @F
@F @F
@T
@BEG_Attrib
3 @RT(0) @RT(0) @RT(0)
@END_Attrib
1 4 @F @F @F @F

@Var @RT(7)sPrefix @RT(0) @T @F @DT @RT(10)STRING(63) @RT(0) @T @T @STRING 0 @F @RT(2)63 @F
@F @F
@T
@BEG_Attrib
3 @RT(0) @RT(0) @RT(0)
@END_Attrib
1 0 @F @F @F @F

@Var @RT(19)mHeatingMoldGeneral @RT(0) @T @T @DERIVED 0 @F @RT(16)tsHeatingGeneral @F
@T
@BEG_Attrib
3 @RT(0) @RT(0) @RT(0)
@END_Attrib
1 0 @F @F @F @F

@Var @RT(21)mHeatingNozzleGeneral @RT(0) @T @T @DERIVED 0 @T @T @DT @RT(22)tyHeatingNozzleGeneral @RT(0) @T @T @UNKNOWN 0 @F
@F @F
@T
@BEG_Attrib
3 @RT(0) @RT(0) @RT(0)
@END_Attrib
1 0 @F @F @F @F

@Var @RT(1)s @RT(0) @T @T @DERIVED 0 @T @T @DT @RT(11)KSYS_Status @RT(0) @T @T @UNKNOWN 0 @F
@F @F
@T
@BEG_Attrib
3 @RT(0) @RT(0) @RT(0)
@END_Attrib
1 0 @F @F @F @F

@Var @RT(5)bEM63 @RT(0) @T @F @DT @RT(4)BOOL @RT(0) @T @T @BASIC 0 @F
@F @F
@T
@BEG_Attrib
3 @RT(0) @RT(0) @RT(0)
@END_Attrib
1 1 @F @F @F @F

@END_Dcl

@END_Export

@BEG_Body
@TL(27)
(**************************************** WARNING ********************************************
 *** The KEBA Kemro K2 System including software is not intended for safety control tasks! ***
 ***                       For further information see Comment tab!                        ***
 *********************************************************************************************)

// mapping from EM83 zone mode (14.6 Table 63) to EM63 zone mode

//    "0" Barrel Zone is not supported    ... EM83: OTHER_0
//    "O" Barrel Zone is off              ... EM83: OFF_1, ONLY_MEASUREMENT_6
//    "A" Barrel Zone is in auto mode     ... EM83: AUTOMATIC_2
//    "T" Barrel Zone is in tuning mode   ... EM83: TUNING_3
//    "S" Barrel Zone is in standby mode  ... EM83: STANDBY_4
//    "M" Barrel Zone is in manual mode   ... EM83: OPEN_LOOP_5

CASE (zoneMode) OF
    nOther_0: fZoneModeToString := "0";
    nOff_1: fZoneModeToString := "O";
    nOnlyMeasurement_6: fZoneModeToString := "O";
    nAutomatic_2: fZoneModeToString := "A";
    nTuning_3: fZoneModeToString := "T";
    nStandby_4: fZoneModeToString := "S";
    nOpenLoop_5: fZoneModeToString := "M";

ELSE
    fZoneModeToString := "0";
END_CASE;

@END_Body

@@@BEG_Comment@@@
@TL(0)

@@@END_Comment@@@

@BEG_Body
@TL(39)
(**************************************** WARNING ********************************************
 *** The KEBA Kemro K2 System including software is not intended for safety control tasks! ***
 ***                       For further information see Comment tab!                        ***
 *********************************************************************************************)

IF (zone.pZoneMode = EMPTY) THEN
   RETURN;
END_IF;

IF (general.piZonesAvailable <> EMPTY) AND (iZoneNr > general.piZonesAvailable^) THEN
    zoneMode := nOther_0;
ELSIF (general.pbHeatingOn <> EMPTY) AND (NOT general.pbHeatingOn^) THEN
    zoneMode := nOff_1;
ELSIF NOT (zone.pbUsed^) THEN
    zoneMode := nOff_1;
ELSIF (zone.pZoneMode^ = enZoneModeDisabled)  THEN
    zoneMode := nOff_1;
ELSIF (zone.pZoneMode^ = enZoneModeMeasure) THEN
    zoneMode := nOnlyMeasurement_6;
ELSIF (zone.pZoneMode^ = enZoneModeConstant) THEN
    zoneMode := nOpenLoop_5;
ELSIF (zone.pbOptimizingActive^) THEN
    zoneMode := nTuning_3;
ELSIF ((general.pbKeepWarmActive <> EMPTY) AND (general.pbKeepWarmActive^)) THEN
    zoneMode := nStandby_4;
ELSE
    zoneMode := nAutomatic_2;
END_IF;

IF (zoneModeEM83 <> zoneMode) THEN
    zoneModeEM83 := zoneMode;
    IF (mbEM63) THEN
       zoneModeEM63 := fZoneModeToString(zoneMode);
    END_IF;
END_IF;

fUpdateHeatingZone := TRUE;

@END_Body

@@@BEG_Comment@@@
@TL(0)

@@@END_Comment@@@

@BEG_Body
@TL(20)
(**************************************** WARNING ********************************************
 *** The KEBA Kemro K2 System including software is not intended for safety control tasks! ***
 ***                       For further information see Comment tab!                        ***
 *********************************************************************************************)

pbLinked := GET_SYNC_REFTO(CONCAT(sPrefix, "Array[", DINT_TO_STRING(iZoneNr),"].bLinked"), T#0s, s);
IF ((pbLinked =EMPTY) OR (NOT pbLinked^)) THEN
    RETURN;
END_IF;

sPrefixZone := CONCAT(sPrefix, DINT_TO_STRING(iZoneNr));
zone.pbOptimizingActive := GET_SYNC_REFTO(CONCAT(sPrefixZone, ".bIsOptimizing"), t#0s, s);
zone.pbEmergencyOperation := GET_SYNC_REFTO(CONCAT(sPrefixZone, ".bEmgOperation"), t#0s, s);

sPrefixZone := CONCAT(sPrefix, "Retain", DINT_TO_STRING(iZoneNr));
zone.pZoneMode := GET_SYNC_REFTO(CONCAT(sPrefixZone, ".ModeVis"), t#0s, s);
zone.pbUsed := GET_SYNC_REFTO(CONCAT(sPrefixZone, ".bUsed"), t#0s, s);

fInitHeatingZone := TRUE;

@END_Body

@@@BEG_Comment@@@
@TL(0)

@@@END_Comment@@@

@BEG_Body
@TL(62)
(**************************************** WARNING ********************************************
 *** The KEBA Kemro K2 System including software is not intended for safety control tasks! ***
 ***                       For further information see Comment tab!                        ***
 *********************************************************************************************)

// SetCfgBrlZn, SetCfgMldZn

IF (NOT bInit) THEN
    mbEM63 := bEM63;
    rtc();
    ts := rtc.CDT;
    bInit := TRUE;
    FOR k := 1 TO cMaxInjectionUnits DO
        sPrefix := CONCAT("HeatingNozzle", DINT_TO_STRING(k));
        mHeatingNozzleGeneral[k].pbKeepWarmActive := GET_SYNC_REFTO(CONCAT(sPrefix, ".sv_bKeepWarmActive"), T#0s, s);
        mHeatingNozzleGeneral[k].pbHeatingOn := GET_SYNC_REFTO(CONCAT(sPrefix, ".sv_bHeatingOn"), T#0s, s);
        mHeatingNozzleGeneral[k].piZonesAvailable := GET_SYNC_REFTO(CONCAT(sPrefix, ".sv_iZonesAvailable"), T#0s, s);
        sPrefix := CONCAT(sPrefix, ".sv_Zone");

        FOR i := 1 TO cMaxHeatingNozzleZones DO
            b := fInitHeatingZone(sPrefix, i, yHeatingZonesNozzle[k, i]);
            IF (NOT b) THEN
               EXIT;
            END_IF;
        END_FOR;
    END_FOR;

    sPrefix := "HeatingMold1.sv_Zone";
    mHeatingMoldGeneral.pbKeepWarmActive := GET_SYNC_REFTO("HeatingMold1.sv_bKeepWarmActive", T#0s, s);
    mHeatingMoldGeneral.pbHeatingOn := GET_SYNC_REFTO("HeatingMold1.sv_bHeatingOn", T#0s, s);
    mHeatingMoldGeneral.piZonesAvailable := GET_SYNC_REFTO("HeatingMold1.sv_iZonesAvailable", T#0s, s);
    FOR i := 1 TO cMaxHeatingMoldZones DO
        b := fInitHeatingZone(sPrefix, i, yHeatingZonesMold[i]);
        IF (NOT b) THEN
            EXIT;
        END_IF;
    END_FOR;

    rtc();
    t := rtc.CDT - ts;

END_IF;

FOR k := 1 TO cMaxInjectionUnits DO
    FOR i := 1 TO cMaxHeatingNozzleZones DO
        b := fUpdateHeatingZone(i, mHeatingNozzleGeneral[k], yHeatingZonesNozzle[k,i], sv_EM63.SetCfgBrlZn[k,i], sv_EM77.SetCfgBrlZn[k,i]);
        IF (NOT b) THEN
           EXIT;
        END_IF;
    END_FOR;
END_FOR;

FOR i := 1 TO cMaxHeatingMoldZones DO
    b := fUpdateHeatingZone(i, mHeatingMoldGeneral, yHeatingZonesMold[i], sv_EM63.SetCfgMldZn[i], sv_EM77.SetCfgMldZn[i]);
    IF (NOT b) THEN
        EXIT;
    END_IF;
END_FOR;

@END_Body

@@@BEG_Comment@@@
@TL(0)

@@@END_Comment@@@
@END_Body

@END_Contents

(* ---- ABProcessDataRecorder.pu ---- *)
(*
@h    ! WARNING !
@h    The Kemro K2 system (including software) only meets category B according to EN 954-1,
@h    thus it is not intended for usage in safety-relevant control applications in the field
@h    of personal safety (e.g. emergency stop).
@h    To implement potentially necessary safety-relevant control tasks, always use additional
@h    external safety devices that are intended for the particular purpose, and meet the necessary
@h    functional safety.
@h    For further information see EN 954-1 (EN ISO 13849-1) and/or the K2-x00 user manual, chapter
@h    "CE conformity, directives and standards".

processdata recorder
*)

IMPORT_OVER_LISTFILE
 FTimeToSec
, KCAT_GetHandle
, KCAT_GetValue
, STOP_PROCESS_ALGORITHM
, GET_SYNC_REFTO
, KCAT_AddValue
, KCAT_RemoveDir
, FGetCatConfigValueString
, CONVERT_LREAL_TO_LWORD
, cCompInjection
, cPDRMaxVars
, KCAT_Type_STRING
, cPDRMaxLines
, tsProcessDataRecorder
, tyyPDRProcessData
, tyyPDRProcessDataRaw
, tevMovementState
, tyPDRConfiguration
, KCAT_HandleData
, KCAT_Status
, tyPDRProcessDataReal
, tyPDRProcessDataRaw
, RTC
, tevMovementStateData
, KSYS_Status
, tsPDRVarRef

END_IMPORT

ALGORITHM_BLOCK ABProcessDataRecorder #DUMMY_EDIT_BLOCK

SYSTEM_VAR
 sv_ProcessDataRecorder : tsProcessDataRecorder;
 sv_iShotCounterAct : DINT;
END_VAR

SYSTEM_OBJECT
 PU_Task_3 : TASK;
 evMovementState : tevMovementState;
 TaskVis : TASK;
 PU_Task_7 : TASK;
END_OBJECT

VAR
 mActProcessData : tyyPDRProcessData;
 mActProcessDataRaw : tyyPDRProcessDataRaw;
 mpiTrigger : REFTO DINT;
 mpiTriggerPU : REFTO DINT;
 mevMovementState : tevMovementState;
 mRecorderConfiguration : tyPDRConfiguration;
 mWriteIdx : DINT;
 mReadIdx : DINT;
 mIdxLastPdrVar : DINT;
 miMode : DINT;
 mpiTriggerClient : REFTO DINT;
END_VAR

VAR CONSTANT
 cConfigNode : STRING(255) := 'Application.ProcessDataRecorder:0';
 cConfigNodeCfgFile : STRING(255) := 'CfgFile';
END_VAR

FUNCTION fReadConfigInt : BOOL
 #DUMMY_EDIT_BLOCK

VAR_INPUT
 name : STRING(255);
END_VAR

VAR_IN_OUT
 value : DINT;
END_VAR

VAR
 handleData : KCAT_HandleData;
 status : KCAT_Status;
END_VAR
#BEGIN_EDIT_BLOCK
fReadConfigInt := FALSE;
handleData := KCAT_GetHandle(CONCAT(cConfigNode, ".", name));
IF (handleData.Status = KCAT_Status_OK) THEN
    status := KCAT_GetValue(handleData.Handle, value);
    IF (status = KCAT_Status_OK) THEN
        fReadConfigInt := TRUE;
    END_IF;
END_IF;

;#END_EDIT_BLOCK END_FUNCTION

FUNCTION fReadConfigString : BOOL
 #DUMMY_EDIT_BLOCK

VAR_INPUT
 name : STRING(255);
END_VAR

VAR_IN_OUT
 value : STRING(255);
END_VAR

VAR
 handleData : KCAT_HandleData;
 status : KCAT_Status;
END_VAR
#BEGIN_EDIT_BLOCK
fReadConfigString := FALSE;
handleData := KCAT_GetHandle(CONCAT(cConfigNode, ".", name));
IF (handleData.Status = KCAT_Status_OK) THEN
    status := KCAT_GetValue(handleData.Handle, value);
    IF (status = KCAT_Status_OK) THEN
        fReadConfigString := TRUE;
    END_IF;
END_IF;

;#END_EDIT_BLOCK END_FUNCTION

FUNCTION fReadOrAddConfigString : BOOL
 #DUMMY_EDIT_BLOCK

VAR_INPUT
 name : STRING(255);
END_VAR

VAR_IN_OUT
 value : STRING(255);
END_VAR

VAR_INPUT
 default : STRING(255);
END_VAR

VAR
 handleData : KCAT_HandleData;
 status : KCAT_Status;
END_VAR
#BEGIN_EDIT_BLOCK
fReadOrAddConfigString := fReadConfigString(name, value);

IF (NOT fReadOrAddConfigString) THEN
        value := default;

        handleData := KCAT_GetHandle(cConfigNode);
        IF (handleData.Status <> KCAT_Status_OK) THEN
            handleData := KCAT_GetRoot();
            handleData := KCAT_AddDir(handleData.Handle, cConfigNode);
        END_IF;
        IF (handleData.Status = KCAT_Status_OK) THEN
            status := KCAT_AddValue(handleData.Handle, name, KCAT_Type_STRING, value);
            fReadOrAddConfigString := status = KCAT_Status_OK;
        END_IF;
END_IF;

;#END_EDIT_BLOCK END_FUNCTION

ALGORITHM aSignalRead

#BEGIN_EDIT_BLOCK
IF (mpiTriggerClient^ = 0) THEN
    IF (mReadIdx <> mWriteIdx) THEN
       IF (miMode = 0) THEN
           // sample mode REAL
          sv_ProcessDataRecorder.data := mActProcessData[mReadIdx + 1];
       ELSIF (miMode = 1) THEN
           // sample mode Raw
          sv_ProcessDataRecorder.dataRaw := mActProcessDataRaw[mReadIdx + 1];
       END_IF;
       mReadIdx := (mReadIdx + 1) MOD cPDRMaxLines;
    END_IF;
END_IF;

;#END_EDIT_BLOCK END_ALGORITHM

ALGORITHM aDoSample

VAR_INPUT
 iGroupId : DINT;
END_VAR

VAR_TEMP
 i : DINT;
END_VAR

VAR
 b : BOOL;
END_VAR
#BEGIN_EDIT_BLOCK
IF (NOT sv_ProcessDataRecorder.bActivate) THEN
    RETURN;
END_IF;
IF (miMode = 0) THEN
    // sample mode REAL
    FOR i := 1 TO mIdxLastPdrVar DO
        IF (mRecorderConfiguration[i].sampleGroup = iGroupId) THEN
            IF (mRecorderConfiguration[i].prReal <> EMPTY) THEN
                mActProcessData[mWriteIdx+1].yParameter[i] := mRecorderConfiguration[i].prReal^;
            ELSIF (mRecorderConfiguration[i].pdTime <> EMPTY) THEN
                mActProcessData[mWriteIdx+1].yParameter[i] := FTimeToSec(mRecorderConfiguration[i].pdTime^);
            ELSIF (mRecorderConfiguration[i].piDInt <> EMPTY) THEN
                mActProcessData[mWriteIdx+1].yParameter[i] := DINT_TO_REAL(mRecorderConfiguration[i].piDInt^);
            END_IF;
        END_IF;
    END_FOR;
ELSIF (miMode = 1) THEN
    // sample mode RAW
     FOR i := 1 TO mIdxLastPdrVar DO
        IF (mRecorderConfiguration[i].sampleGroup = iGroupId) THEN
            CASE (mRecorderConfiguration[i].nType) OF
                cPDRVarTypeReal:
                    b := CONVERT_LREAL_TO_LWORD(REAL_TO_LREAL(mRecorderConfiguration[i].prReal^), mActProcessDataRaw[mWriteIdx+1].yParameter[i]);

                cPDRVarTypeTime:
                    mActProcessDataRaw[mWriteIdx+1].yParameter[i] := LINT_TO_LWORD(TIME_TO_LINT(mRecorderConfiguration[i].pdTime^));

                cPDRVarTypeDInt:
                    mActProcessDataRaw[mWriteIdx+1].yParameter[i] := LINT_TO_LWORD(DINT_TO_LINT(mRecorderConfiguration[i].piDInt^));

                cPDRVarTypeLReal:
                    b := CONVERT_LREAL_TO_LWORD(mRecorderConfiguration[i].prLReal^, mActProcessDataRaw[mWriteIdx+1].yParameter[i]);

                cPDRVarTypeBool:
                    mActProcessDataRaw[mWriteIdx+1].yParameter[i] := LINT_TO_LWORD(BOOL_TO_LINT(mRecorderConfiguration[i].pbBool^));

                cPDRVarTypeDT:
                    mActProcessDataRaw[mWriteIdx+1].yParameter[i] := LINT_TO_LWORD(DATE_TO_LINT(DT_TO_DATE(mRecorderConfiguration[i].pdDT^))+TIME_TO_LINT(TOD_TO_TIME(DT_TO_TOD(mRecorderConfiguration[i].pdDT^))));

                cPDRVarTypeSInt:
                    mActProcessDataRaw[mWriteIdx+1].yParameter[i] := LINT_TO_LWORD(SINT_TO_LINT(mRecorderConfiguration[i].piSInt^));

                cPDRVarTypeInt:
                    mActProcessDataRaw[mWriteIdx+1].yParameter[i] := LINT_TO_LWORD(INT_TO_LINT(mRecorderConfiguration[i].piInt^));

                cPDRVarTypeLInt:
                    mActProcessDataRaw[mWriteIdx+1].yParameter[i] := LINT_TO_LWORD(mRecorderConfiguration[i].piLInt^);

                cPDRVarTypeUSInt:
                    mActProcessDataRaw[mWriteIdx+1].yParameter[i] := USINT_TO_LWORD(mRecorderConfiguration[i].piUSInt^);

                cPDRVarTypeUInt:
                    mActProcessDataRaw[mWriteIdx+1].yParameter[i] := UINT_TO_LWORD(mRecorderConfiguration[i].piUInt^);

                cPDRVarTypeUDInt:
                    mActProcessDataRaw[mWriteIdx+1].yParameter[i] := UDINT_TO_LWORD(mRecorderConfiguration[i].piUDInt^);

                cPDRVarTypeULInt:
                    mActProcessDataRaw[mWriteIdx+1].yParameter[i] := ULINT_TO_LWORD(mRecorderConfiguration[i].piULInt^);

             END_CASE;
        END_IF;
    END_FOR;
END_IF;

;#END_EDIT_BLOCK END_ALGORITHM

(*
@h    ! WARNING !
@h    The Kemro K2 system (including software) only meets category B according to EN 954-1,
@h    thus it is not intended for usage in safety-relevant control applications in the field
@h    of personal safety (e.g. emergency stop).
@h    To implement potentially necessary safety-relevant control tasks, always use additional
@h    external safety devices that are intended for the particular purpose, and meet the necessary
@h    functional safety.
@h    For further information see EN 954-1 (EN ISO 13849-1) and/or the K2-x00 user manual, chapter
@h    "CE conformity, directives and standards".

*)

POSTUPDATE_ALGORITHM pTriggerVariable ON PU_Task_3 WITH mpiTriggerPU^

VAR
 fbRtc : RTC;
 t : TIME;
 ts : TIME;
END_VAR

VAR CONSTANT
 emptyProcessData : tyPDRProcessDataReal;
 emptyProcessDataRaw : tyPDRProcessDataRaw;
END_VAR
#BEGIN_EDIT_BLOCK
(**************************************** WARNING ********************************************
 *** The KEBA Kemro K2 System including software is not intended for safety control tasks! ***
 ***                       For further information see Comment tab!                        ***
 *********************************************************************************************)

ts := GET_RUNTIME();
aDoSample(0);
fbRtc();

IF (miMode = 0) THEN
    // sample mode REAL
    mActProcessData[mWriteIdx+1].iTrigger := mpiTriggerPU^;
    mActProcessData[mWriteIdx+1].dTimeStamp := fbRtc.CDT;
    mWriteIdx := (mWriteIdx + 1) MOD cPDRMaxLines;
    mActProcessData[mWriteIdx + 1].yParameter := emptyProcessData;
    mActProcessData[mWriteIdx + 1].iTrigger := 0;
ELSIF (miMode = 1) THEN
    // sample mode RAW
    mActProcessDataRaw[mWriteIdx+1].iTrigger := mpiTriggerPU^;
    mActProcessDataRaw[mWriteIdx+1].dTimeStamp := fbRtc.CDT;
    mWriteIdx := (mWriteIdx + 1) MOD cPDRMaxLines;
    mActProcessDataRaw[mWriteIdx + 1].yParameter := emptyProcessDataRaw;
    mActProcessDataRaw[mWriteIdx + 1].iTrigger := 0;
END_IF;

IF (mWriteIdx = mReadIdx) THEN
    mReadIdx := (mReadIdx + 1) MOD cPDRMaxLines;
END_IF;

aSignalRead();

t := GET_RUNTIME() - ts;

;#END_EDIT_BLOCK END_ALGORITHM

(*
@h    ! WARNING !
@h    The Kemro K2 system (including software) only meets category B according to EN 954-1,
@h    thus it is not intended for usage in safety-relevant control applications in the field
@h    of personal safety (e.g. emergency stop).
@h    To implement potentially necessary safety-relevant control tasks, always use additional
@h    external safety devices that are intended for the particular purpose, and meet the necessary
@h    functional safety.
@h    For further information see EN 954-1 (EN ISO 13849-1) and/or the K2-x00 user manual, chapter
@h    "CE conformity, directives and standards".

collects processdata: sample values at inject
*)

EVENT_ALGORITHM pInjectData ON PU_Task_3 WITH mevMovementState

VAR_INPUT
 evMovementStateData : tevMovementStateData;
END_VAR
#BEGIN_EDIT_BLOCK
(**************************************** WARNING ********************************************
 *** The KEBA Kemro K2 System including software is not intended for safety control tasks! ***
 ***                       For further information see Comment tab!                        ***
 *********************************************************************************************)

IF ((evMovementStateData.DeviceId.CompId = cCompInjection)
   AND (evMovementStateData.DeviceId.IndexId = 1)
   AND (evMovementStateData.MoveId   = cMoveInject)
   AND (evMovementStateData.MoveDir  = cMoveFwd)
   AND (evMovementStateData.State  = nActive)) THEN

    // copy data at inject time
    aDoSample(16);
END_IF;

;#END_EDIT_BLOCK END_ALGORITHM

ALGORITHM aInit

VAR_TEMP
 activate : DINT;
 i : DINT;
END_VAR

VAR
 b : BOOL;
 name : STRING(255);
 s : KSYS_Status;
 cnt : INT;
 cfgFile : STRING(255);
END_VAR
#BEGIN_EDIT_BLOCK
b := fReadOrAddConfigString(cConfigNodeCfgFile, cfgFile, 'workspace/data/pdr.cfg');

miMode := 0;
b := fReadConfigInt("Mode", miMode);
b := fReadConfigInt("Activate", activate);

IF (fReadConfigString("Trigger", name)) THEN
   mpiTrigger := GET_SYNC_REFTO(name, T#0s, s);
END_IF;

IF (mpiTrigger = EMPTY) THEN
    mpiTrigger := @sv_iShotCounterAct;
END_IF;

FOR i := 1 TO cPDRMaxVars DO
   mRecorderConfiguration[i].nType := cPDRVarTypeNone;
   IF (fReadConfigString(CONCAT("Var:", DINT_TO_STRING(i), ".Name"), name)) THEN

       /////////   R E A L   /////////
       IF (mRecorderConfiguration[i].nType = cPDRVarTypeNone) THEN
          mRecorderConfiguration[i].prReal := GET_SYNC_REFTO(name, T#0s, s);
          IF (s = KSYS_Status_OK) THEN
             mRecorderConfiguration[i].nType := cPDRVarTypeReal;
          END_IF;
       END_IF;
       /////////   T I M E   /////////
       IF (mRecorderConfiguration[i].nType = cPDRVarTypeNone) THEN
          mRecorderConfiguration[i].pdTime := GET_SYNC_REFTO(name, T#0s, s);
          IF (s = KSYS_Status_OK) THEN
             mRecorderConfiguration[i].nType := cPDRVarTypeTime;
          END_IF;
       END_IF;
       /////////   D I N T   /////////
       IF (mRecorderConfiguration[i].nType = cPDRVarTypeNone) THEN
          mRecorderConfiguration[i].piDInt := GET_SYNC_REFTO(name, T#0s, s);
          IF (s = KSYS_Status_OK) THEN
             mRecorderConfiguration[i].nType := cPDRVarTypeDInt;
          END_IF;
       END_IF;

       IF (miMode > 0) THEN
            /////////   L R E A L   /////////
            IF (mRecorderConfiguration[i].nType = cPDRVarTypeNone) THEN
                mRecorderConfiguration[i].prLReal := GET_SYNC_REFTO(name, T#0s, s);
                IF (s = KSYS_Status_OK) THEN
                    mRecorderConfiguration[i].nType := cPDRVarTypeLReal;
                END_IF;
            END_IF;
            /////////   B O O L   /////////
            IF (mRecorderConfiguration[i].nType = cPDRVarTypeNone) THEN
                mRecorderConfiguration[i].pbBool := GET_SYNC_REFTO(name, T#0s, s);
                IF (s = KSYS_Status_OK) THEN
                    mRecorderConfiguration[i].nType := cPDRVarTypeBool;
                END_IF;
            END_IF;
            /////////   D A T E  &  T I M E   /////////
            IF (mRecorderConfiguration[i].nType = cPDRVarTypeNone) THEN
                mRecorderConfiguration[i].pdDT := GET_SYNC_REFTO(name, T#0s, s);
                IF (s = KSYS_Status_OK) THEN
                    mRecorderConfiguration[i].nType := cPDRVarTypeDT;
                END_IF;
            END_IF;
            /////////   S I N T   /////////
            IF (mRecorderConfiguration[i].nType = cPDRVarTypeNone) THEN
                mRecorderConfiguration[i].piSInt := GET_SYNC_REFTO(name, T#0s, s);
                IF (s = KSYS_Status_OK) THEN
                    mRecorderConfiguration[i].nType := cPDRVarTypeSInt;
                END_IF;
            END_IF;
            /////////   I N T   /////////
            IF (mRecorderConfiguration[i].nType = cPDRVarTypeNone) THEN
                mRecorderConfiguration[i].piInt := GET_SYNC_REFTO(name, T#0s, s);
                IF (s = KSYS_Status_OK) THEN
                    mRecorderConfiguration[i].nType := cPDRVarTypeInt;
                END_IF;
            END_IF;
            /////////   L I N T   /////////
            IF (mRecorderConfiguration[i].nType = cPDRVarTypeNone) THEN
                mRecorderConfiguration[i].piLInt := GET_SYNC_REFTO(name, T#0s, s);
                IF (s = KSYS_Status_OK) THEN
                    mRecorderConfiguration[i].nType := cPDRVarTypeLInt;
                END_IF;
            END_IF;
            /////////   U S I N T   /////////
            IF (mRecorderConfiguration[i].nType = cPDRVarTypeNone) THEN
                mRecorderConfiguration[i].piUSInt := GET_SYNC_REFTO(name, T#0s, s);
                IF (s = KSYS_Status_OK) THEN
                    mRecorderConfiguration[i].nType := cPDRVarTypeUSInt;
                END_IF;
            END_IF;
                /////////   U I N T   /////////
            IF (mRecorderConfiguration[i].nType = cPDRVarTypeNone) THEN
                mRecorderConfiguration[i].piUInt := GET_SYNC_REFTO(name, T#0s, s);
                IF (s = KSYS_Status_OK) THEN
                    mRecorderConfiguration[i].nType := cPDRVarTypeUInt;
                END_IF;
            END_IF;
            /////////   U D I N T   /////////
            IF (mRecorderConfiguration[i].nType = cPDRVarTypeNone) THEN
                mRecorderConfiguration[i].piUDInt := GET_SYNC_REFTO(name, T#0s, s);
                IF (s = KSYS_Status_OK) THEN
                    mRecorderConfiguration[i].nType := cPDRVarTypeUDInt;
                END_IF;
            END_IF;
            /////////   U L I N T   /////////
            IF (mRecorderConfiguration[i].nType = cPDRVarTypeNone) THEN
                mRecorderConfiguration[i].piULInt := GET_SYNC_REFTO(name, T#0s, s);
                IF (s = KSYS_Status_OK) THEN
                    mRecorderConfiguration[i].nType := cPDRVarTypeULInt;
                END_IF;
            END_IF;
       END_IF;

       // Type found ... save last used index in configuration
       IF (mRecorderConfiguration[i].nType <> cPDRVarTypeNone) THEN
          mIdxLastPdrVar := i;
       END_IF;

       cnt := cnt + 1;
       b := fReadConfigInt(CONCAT("Var:", DINT_TO_STRING(i), ".SampleGroup"), mRecorderConfiguration[i].sampleGroup);
   END_IF;
   sv_ProcessDataRecorder.yActiveVariables[i] := mRecorderConfiguration[i].nType;
END_FOR;

IF (activate <> 0) THEN
    sv_ProcessDataRecorder.bActivate := TRUE;
END_IF;

;#END_EDIT_BLOCK END_ALGORITHM

PROCESS_ALGORITHM paInit ON TaskVis(1) AUTOSTART

#BEGIN_EDIT_BLOCK
STOP_PROCESS_ALGORITHM();

aInit();

;#END_EDIT_BLOCK END_ALGORITHM

POSTUPDATE_ALGORITHM pReadDone ON PU_Task_3 WITH mpiTriggerClient^

#BEGIN_EDIT_BLOCK
aSignalRead();

;#END_EDIT_BLOCK END_ALGORITHM

POSTUPDATE_ALGORITHM pActivate ON PU_Task_7 WITH sv_ProcessDataRecorder.bActivate

#BEGIN_EDIT_BLOCK
IF (sv_ProcessDataRecorder.bActivate) THEN
   mpiTriggerPU := mpiTrigger;
   mevMovementState := evMovementState;
   IF (miMode = 0) THEN
       // sample mode real
       mpiTriggerClient := @sv_ProcessDataRecorder.data.iTrigger;
   ELSIF (miMode = 1) THEN
       // sample mode raw
       mpiTriggerClient := @sv_ProcessDataRecorder.dataRaw.iTrigger;
   END_IF;
ELSE
   mpiTriggerPU := EMPTY;
   mevMovementState := EMPTY;
   mpiTriggerClient := EMPTY;
END_IF;

;#END_EDIT_BLOCK END_ALGORITHM

POSTUPDATE_ALGORITHM pReload ON TaskVis WITH sv_ProcessDataRecorder.iReloadConfiguration

VAR_TEMP
 i : DINT;
END_VAR

VAR
 b : BOOL;
 s : KCAT_Status;
 handleData : KCAT_HandleData;
 cfgFile : STRING(255);
 workPath : STRING(255);
END_VAR

VAR CONSTANT
 emptyElem : tsPDRVarRef;
END_VAR
#BEGIN_EDIT_BLOCK
IF (sv_ProcessDataRecorder.iReloadConfiguration MOD 2 = 1) THEN
    sv_ProcessDataRecorder.bActivate := FALSE;

    cfgFile := "";
    b := fReadConfigString(cConfigNodeCfgFile, cfgFile);
    handleData := KCAT_GetHandle(cConfigNode);
    IF (handleData.Status = KCAT_Status_OK) THEN
        s := KCAT_RemoveDir(handleData.Handle);
    END_IF;

    workPath := FGetCatConfigValueString("System.workPath", "/");

    FOR i := 1 TO cPDRMaxVars DO
        mRecorderConfiguration[i] := emptyElem;
    END_FOR;

    mWriteIdx := 0;
    mReadIdx := 0;

    s := KCAT_Load(CONCAT(workPath, "/", cfgFile));

    aInit();

    IF (LEN(cfgFile) > 0) THEN
      b := fReadOrAddConfigString(cConfigNodeCfgFile, cfgFile, cfgFile);
    END_IF;

    sv_ProcessDataRecorder.iReloadConfiguration := sv_ProcessDataRecorder.iReloadConfiguration + 1;
END_IF;

;#END_EDIT_BLOCK END_ALGORITHM

END_ALGORITHM_BLOCK

#END_OF_IEC_PART

@Puma @IecEditor 6 68 @Pou 25
@@@BEG_Comment@@@
@h    ! WARNING !
@h    The Kemro K2 system (including software) only meets category B according to EN 954-1,
@h    thus it is not intended for usage in safety-relevant control applications in the field
@h    of personal safety (e.g. emergency stop).
@h    To implement potentially necessary safety-relevant control tasks, always use additional
@h    external safety devices that are intended for the particular purpose, and meet the necessary
@h    functional safety.
@h    For further information see EN 954-1 (EN ISO 13849-1) and/or the K2-x00 user manual, chapter
@h    "CE conformity, directives and standards".

processdata recorder
@@@END_Comment@@@

@BEG_Contents

@BEG_Func
@RT(17)FuncTreeContainer
9
@Var @RT(10)FTimeToSec @RT(0) @T @T @DERIVED 0 @F @RT(8)FUNCTION @F
@T
@BEG_Attrib
0 @RT(0) @RT(0)
@END_Attrib
1 1 @F @F @F @F

@Var @RT(14)KCAT_GetHandle @RT(0) @T @T @DERIVED 0 @F @RT(22)KEBA_STANDARD_FUNCTION @F
@T
@BEG_Attrib
0 @RT(0) @RT(0)
@END_Attrib
1 1 @F @F @F @F

@Var @RT(13)KCAT_GetValue @RT(0) @T @T @DERIVED 0 @F @RT(22)KEBA_STANDARD_FUNCTION @F
@T
@BEG_Attrib
0 @RT(0) @RT(0)
@END_Attrib
1 1 @F @F @F @F

@Var @RT(22)STOP_PROCESS_ALGORITHM @RT(0) @T @T @DERIVED 0 @F @RT(23)KEBA_STANDARD_PROCEDURE @F
@T
@BEG_Attrib
0 @RT(0) @RT(0)
@END_Attrib
1 1 @F @F @F @F

@Var @RT(14)GET_SYNC_REFTO @RT(0) @T @T @DERIVED 0 @F @RT(22)KEBA_STANDARD_FUNCTION @F
@T
@BEG_Attrib
0 @RT(0) @RT(0)
@END_Attrib
1 1 @F @F @F @F

@Var @RT(13)KCAT_AddValue @RT(0) @T @T @DERIVED 0 @F @RT(22)KEBA_STANDARD_FUNCTION @F
@T
@BEG_Attrib
0 @RT(0) @RT(0)
@END_Attrib
1 1 @F @F @F @F

@Var @RT(14)KCAT_RemoveDir @RT(0) @T @T @DERIVED 0 @F @RT(22)KEBA_STANDARD_FUNCTION @F
@T
@BEG_Attrib
0 @RT(0) @RT(0)
@END_Attrib
1 1 @F @F @F @F

@Var @RT(24)FGetCatConfigValueString @RT(0) @T @T @DERIVED 0 @F @RT(8)FUNCTION @F
@T
@BEG_Attrib
0 @RT(0) @RT(0)
@END_Attrib
1 1 @F @F @F @F

@Var @RT(22)CONVERT_LREAL_TO_LWORD @RT(0) @T @T @DERIVED 0 @F @RT(22)KEBA_STANDARD_FUNCTION @F
@T
@BEG_Attrib
0 @RT(0) @RT(0)
@END_Attrib
1 1 @F @F @F @F

@END_Func

@BEG_Const
@RT(18)ConstTreeContainer
4
@Var @RT(14)cCompInjection @RT(0) @T @F @DT @RT(4)DINT @RT(0) @T @T @BASIC 0 @F
@F @F
@T
@BEG_Attrib
0 @RT(3)104 @RT(19)Component Injection
@END_Attrib
1 1 @F @F @F @F

@Var @RT(11)cPDRMaxVars @RT(0) @T @F @DT @RT(4)DINT @RT(0) @T @T @BASIC 0 @F
@F @F
@T
@BEG_Attrib
0 @RT(3)128 @RT(0)
@END_Attrib
1 1 @F @F @F @F

@Var @RT(16)KCAT_Type_STRING @RT(0) @T @T @DERIVED 0 @F @RT(9)KCAT_Type @F
@T
@BEG_Attrib
0 @RT(1)3 @RT(0)
@END_Attrib
1 1 @F @F @F @F

@Var @RT(12)cPDRMaxLines @RT(0) @T @F @DT @RT(4)DINT @RT(0) @T @T @BASIC 0 @F
@F @F
@T
@BEG_Attrib
0 @RT(2)10 @RT(0)
@END_Attrib
1 1 @F @F @F @F

@END_Const

@BEG_Export

@BEG_Kind
@ALGORITHM_BLOCK @RT(21)ABProcessDataRecorder @STRUCTURED_TEXT
@RT(0) @RT(0) @RT(0)
@END_Kind

@BEG_Dcl
@RT(16)DclTreeContainer
19
@Var @RT(22)sv_ProcessDataRecorder @RT(0) @T @T @DERIVED 0 @T @T @DT @RT(21)tsProcessDataRecorder @RT(0) @T @T @UNKNOWN 0 @F
@F @F
@T
@BEG_Attrib
3 @RT(0) @RT(0) @RT(0)
@END_Attrib
1 8 @F @F @F @F

@Var @RT(18)sv_iShotCounterAct @RT(0) @T @F @DT @RT(4)DINT @RT(0) @T @T @BASIC 0 @F
@F @F
@T
@BEG_Attrib
3 @RT(0) @RT(0) @RT(0)
@END_Attrib
1 8 @F @F @F @F

@Var @RT(9)PU_Task_3 @RT(0) @T @F @DT @RT(4)TASK @RT(0) @T @T @BASIC 0 @F
@F @F
@T
@BEG_Attrib
3 @RT(0) @RT(0) @RT(0)
@END_Attrib
1 7 @F @F @F @F

@Var @RT(15)mActProcessData @RT(0) @T @T @DERIVED 0 @T @T @DT @RT(17)tyyPDRProcessData @RT(0) @T @T @UNKNOWN 0 @F
@F @F
@T
@BEG_Attrib
3 @RT(0) @RT(0) @RT(0)
@END_Attrib
1 0 @F @F @F @F

@Var @RT(18)mActProcessDataRaw @RT(0) @T @T @DERIVED 0 @T @T @DT @RT(20)tyyPDRProcessDataRaw @RT(0) @T @T @UNKNOWN 0 @F
@F @F
@T
@BEG_Attrib
3 @RT(0) @RT(0) @RT(0)
@END_Attrib
1 0 @F @F @F @F

@Var @RT(15)evMovementState @RT(0) @T @T @DERIVED 0 @T @T @DT @RT(16)tevMovementState @RT(0) @T @T @UNKNOWN 0 @F
@F @F
@T
@BEG_Attrib
3 @RT(0) @RT(0) @RT(0)
@END_Attrib
1 7 @F @F @F @F

@Var @RT(11)cConfigNode @RT(0) @T @F @DT @RT(11)STRING(255) @RT(0) @T @T @STRING 0 @F @RT(3)255 @F
@F @F
@T
@BEG_Attrib
3 @RT(35)'Application.ProcessDataRecorder:0' @RT(0) @RT(0)
@END_Attrib
1 15 @F @F @F @F

@Var @RT(18)cConfigNodeCfgFile @RT(0) @T @F @DT @RT(11)STRING(255) @RT(0) @T @T @STRING 0 @F @RT(3)255 @F
@F @F
@T
@BEG_Attrib
3 @RT(9)'CfgFile' @RT(0) @RT(0)
@END_Attrib
1 15 @F @F @F @F

@Var @RT(10)mpiTrigger @RT(0) @T @T @REFTO 0 @T @DT @RT(4)DINT @RT(0) @T @T @BASIC 0 @F
@F @F
@T
@BEG_Attrib
3 @RT(0) @RT(0) @RT(0)
@END_Attrib
1 0 @F @F @F @F

@Var @RT(12)mpiTriggerPU @RT(0) @T @T @REFTO 0 @T @DT @RT(4)DINT @RT(0) @T @T @BASIC 0 @F
@F @F
@T
@BEG_Attrib
3 @RT(0) @RT(0) @RT(0)
@END_Attrib
1 0 @F @F @F @F

@Var @RT(7)TaskVis @RT(0) @T @T @RENAMED 0 @T @T @DT @RT(4)TASK @RT(0) @T @T @BASIC 0 @F
@F @F
@T
@BEG_Attrib
3 @RT(0) @RT(0) @RT(0)
@END_Attrib
1 7 @F @F @F @F

@Var @RT(16)mevMovementState @RT(0) @T @T @DERIVED 0 @T @T @DT @RT(16)tevMovementState @RT(0) @T @T @UNKNOWN 0 @F
@F @F
@T
@BEG_Attrib
3 @RT(0) @RT(0) @RT(0)
@END_Attrib
1 0 @F @F @F @F

@Var @RT(22)mRecorderConfiguration @RT(0) @T @T @DERIVED 0 @T @T @DT @RT(18)tyPDRConfiguration @RT(0) @T @T @UNKNOWN 0 @F
@F @F
@T
@BEG_Attrib
3 @RT(0) @RT(0) @RT(0)
@END_Attrib
1 0 @F @F @F @F

@Var @RT(9)mWriteIdx @RT(0) @T @F @DT @RT(4)DINT @RT(0) @T @T @BASIC 0 @F
@F @F
@T
@BEG_Attrib
3 @RT(0) @RT(0) @RT(0)
@END_Attrib
1 0 @F @F @F @F

@Var @RT(8)mReadIdx @RT(0) @T @F @DT @RT(4)DINT @RT(0) @T @T @BASIC 0 @F
@F @F
@T
@BEG_Attrib
3 @RT(0) @RT(0) @RT(0)
@END_Attrib
1 0 @F @F @F @F

@Var @RT(9)PU_Task_7 @RT(0) @T @T @RENAMED 0 @T @T @DT @RT(4)TASK @RT(0) @T @T @BASIC 0 @F
@F @F
@T
@BEG_Attrib
3 @RT(0) @RT(0) @RT(0)
@END_Attrib
1 7 @F @F @F @F

@Var @RT(14)mIdxLastPdrVar @RT(0) @T @F @DT @RT(4)DINT @RT(0) @T @T @BASIC 0 @F
@F @F
@T
@BEG_Attrib
3 @RT(0) @RT(0) @RT(0)
@END_Attrib
1 0 @F @F @F @F

@Var @RT(6)miMode @RT(0) @T @F @DT @RT(4)DINT @RT(0) @T @T @BASIC 0 @F
@F @F
@T
@BEG_Attrib
3 @RT(0) @RT(0) @RT(0)
@END_Attrib
1 0 @F @F @F @F

@Var @RT(16)mpiTriggerClient @RT(0) @T @T @REFTO 0 @T @DT @RT(4)DINT @RT(0) @T @T @BASIC 0 @F
@F @F
@T
@BEG_Attrib
3 @RT(0) @RT(0) @RT(0)
@END_Attrib
1 0 @F @F @F @F

@END_Dcl

@END_Export

@BEG_Body

12

@BEG_Export

@BEG_Algo
@FUNCTION @RT(14)fReadConfigInt @STRUCTURED_TEXT
@RT(4)BOOL @RT(0) @RT(0) @F @F
@END_Algo

@BEG_Dcl
@RT(16)DclTreeContainer
4
@Var @RT(4)name @RT(0) @T @F @DT @RT(11)STRING(255) @RT(0) @T @T @STRING 0 @F @RT(3)255 @F
@F @F
@T
@BEG_Attrib
3 @RT(0) @RT(0) @RT(0)
@END_Attrib
1 1 @F @F @F @F

@Var @RT(5)value @RT(0) @T @F @DT @RT(4)DINT @RT(0) @T @T @BASIC 0 @F
@F @F
@T
@BEG_Attrib
3 @RT(0) @RT(0) @RT(0)
@END_Attrib
1 2 @F @F @F @F

@Var @RT(10)handleData @RT(0) @T @T @DERIVED 0 @T @T @DT @RT(15)KCAT_HandleData @RT(0) @T @T @UNKNOWN 0 @F
@F @F
@T
@BEG_Attrib
3 @RT(0) @RT(0) @RT(0)
@END_Attrib
1 0 @F @F @F @F

@Var @RT(6)status @RT(0) @T @T @DERIVED 0 @T @T @DT @RT(11)KCAT_Status @RT(0) @T @T @UNKNOWN 0 @F
@F @F
@T
@BEG_Attrib
3 @RT(0) @RT(0) @RT(0)
@END_Attrib
1 0 @F @F @F @F

@END_Dcl

@END_Export

@BEG_Export

@BEG_Algo
@FUNCTION @RT(17)fReadConfigString @STRUCTURED_TEXT
@RT(4)BOOL @RT(0) @RT(0) @F @F
@END_Algo

@BEG_Dcl
@RT(16)DclTreeContainer
4
@Var @RT(4)name @RT(0) @T @F @DT @RT(11)STRING(255) @RT(0) @T @T @STRING 0 @F @RT(3)255 @F
@F @F
@T
@BEG_Attrib
3 @RT(0) @RT(0) @RT(0)
@END_Attrib
1 1 @F @F @F @F

@Var @RT(5)value @RT(0) @T @F @DT @RT(11)STRING(255) @RT(0) @T @T @STRING 0 @F @RT(3)255 @F
@F @F
@T
@BEG_Attrib
3 @RT(0) @RT(0) @RT(0)
@END_Attrib
1 2 @F @F @F @F

@Var @RT(10)handleData @RT(0) @T @T @DERIVED 0 @T @T @DT @RT(15)KCAT_HandleData @RT(0) @T @T @UNKNOWN 0 @F
@F @F
@T
@BEG_Attrib
3 @RT(0) @RT(0) @RT(0)
@END_Attrib
1 0 @F @F @F @F

@Var @RT(6)status @RT(0) @T @T @DERIVED 0 @T @T @DT @RT(11)KCAT_Status @RT(0) @T @T @UNKNOWN 0 @F
@F @F
@T
@BEG_Attrib
3 @RT(0) @RT(0) @RT(0)
@END_Attrib
1 0 @F @F @F @F

@END_Dcl

@END_Export

@BEG_Export

@BEG_Algo
@FUNCTION @RT(22)fReadOrAddConfigString @STRUCTURED_TEXT
@RT(4)BOOL @RT(0) @RT(0) @F @F
@END_Algo

@BEG_Dcl
@RT(16)DclTreeContainer
5
@Var @RT(4)name @RT(0) @T @F @DT @RT(11)STRING(255) @RT(0) @T @T @STRING 0 @F @RT(3)255 @F
@F @F
@T
@BEG_Attrib
3 @RT(0) @RT(0) @RT(0)
@END_Attrib
1 1 @F @F @F @F

@Var @RT(5)value @RT(0) @T @F @DT @RT(11)STRING(255) @RT(0) @T @T @STRING 0 @F @RT(3)255 @F
@F @F
@T
@BEG_Attrib
3 @RT(0) @RT(0) @RT(0)
@END_Attrib
1 2 @F @F @F @F

@Var @RT(10)handleData @RT(0) @T @T @DERIVED 0 @T @T @DT @RT(15)KCAT_HandleData @RT(0) @T @T @UNKNOWN 0 @F
@F @F
@T
@BEG_Attrib
3 @RT(0) @RT(0) @RT(0)
@END_Attrib
1 0 @F @F @F @F

@Var @RT(6)status @RT(0) @T @T @DERIVED 0 @T @T @DT @RT(11)KCAT_Status @RT(0) @T @T @UNKNOWN 0 @F
@F @F
@T
@BEG_Attrib
3 @RT(0) @RT(0) @RT(0)
@END_Attrib
1 0 @F @F @F @F

@Var @RT(7)default @RT(0) @T @F @DT @RT(11)STRING(255) @RT(0) @T @T @STRING 0 @F @RT(3)255 @F
@F @F
@T
@BEG_Attrib
3 @RT(0) @RT(0) @RT(0)
@END_Attrib
1 1 @F @F @F @F

@END_Dcl

@END_Export

@BEG_Export

@BEG_Algo
@ALGORITHM @RT(11)aSignalRead @STRUCTURED_TEXT
@RT(0) @RT(0) @RT(0) @F @F
@END_Algo

@BEG_Dcl
@RT(16)DclTreeContainer
0
@END_Dcl

@END_Export

@BEG_Export

@BEG_Algo
@ALGORITHM @RT(9)aDoSample @STRUCTURED_TEXT
@RT(0) @RT(0) @RT(0) @F @F
@END_Algo

@BEG_Dcl
@RT(16)DclTreeContainer
3
@Var @RT(8)iGroupId @RT(0) @T @F @DT @RT(4)DINT @RT(0) @T @T @BASIC 0 @F
@F @F
@T
@BEG_Attrib
3 @RT(0) @RT(0) @RT(0)
@END_Attrib
1 1 @F @F @F @F

@Var @RT(1)i @RT(0) @T @F @DT @RT(4)DINT @RT(0) @T @T @BASIC 0 @F
@F @F
@T
@BEG_Attrib
3 @RT(0) @RT(0) @RT(0)
@END_Attrib
1 4 @F @F @F @F

@Var @RT(1)b @RT(0) @T @F @DT @RT(4)BOOL @RT(0) @T @T @BASIC 0 @F
@F @F
@T
@BEG_Attrib
3 @RT(0) @RT(0) @RT(0)
@END_Attrib
1 0 @F @F @F @F

@END_Dcl

@END_Export

@BEG_Export

@BEG_Algo
@POSTUPDATE_ALGORITHM @RT(16)pTriggerVariable @STRUCTURED_TEXT
@RT(0) @RT(13)mpiTriggerPU^ @RT(9)PU_Task_3 @F @F
@END_Algo

@BEG_Dcl
@RT(16)DclTreeContainer
5
@Var @RT(16)emptyProcessData @RT(0) @T @T @DERIVED 0 @T @T @DT @RT(20)tyPDRProcessDataReal @RT(0) @T @T @UNKNOWN 0 @F
@F @F
@T
@BEG_Attrib
3 @RT(0) @RT(0) @RT(0)
@END_Attrib
1 15 @F @F @F @F

@Var @RT(19)emptyProcessDataRaw @RT(0) @T @T @DERIVED 0 @T @T @DT @RT(19)tyPDRProcessDataRaw @RT(0) @T @T @UNKNOWN 0 @F
@F @F
@T
@BEG_Attrib
3 @RT(0) @RT(0) @RT(0)
@END_Attrib
1 15 @F @F @F @F

@Var @RT(5)fbRtc @RT(0) @T @T @DERIVED 0 @T @T @DT @RT(3)RTC @RT(0) @T @T @UNKNOWN 0 @F
@F @F
@T
@BEG_Attrib
3 @RT(0) @RT(0) @RT(0)
@END_Attrib
1 0 @F @F @F @F

@Var @RT(1)t @RT(0) @T @F @DT @RT(4)TIME @RT(0) @T @T @BASIC 0 @F
@F @F
@T
@BEG_Attrib
3 @RT(0) @RT(0) @RT(0)
@END_Attrib
1 0 @F @F @F @F

@Var @RT(2)ts @RT(0) @T @F @DT @RT(4)TIME @RT(0) @T @T @BASIC 0 @F
@F @F
@T
@BEG_Attrib
3 @RT(0) @RT(0) @RT(0)
@END_Attrib
1 0 @F @F @F @F

@END_Dcl

@END_Export

@BEG_Export

@BEG_Algo
@EVENT_ALGORITHM @RT(11)pInjectData @STRUCTURED_TEXT
@RT(0) @RT(16)mevMovementState @RT(9)PU_Task_3 @F @F
@END_Algo

@BEG_Dcl
@RT(16)DclTreeContainer
1
@Var @RT(19)evMovementStateData @RT(0) @T @T @DERIVED 0 @T @T @DT @RT(20)tevMovementStateData @RT(0) @T @T @UNKNOWN 0 @F
@F @F
@T
@BEG_Attrib
3 @RT(0) @RT(0) @RT(0)
@END_Attrib
1 1 @F @F @F @F

@END_Dcl

@END_Export

@BEG_Export

@BEG_Algo
@ALGORITHM @RT(5)aInit @STRUCTURED_TEXT
@RT(0) @RT(0) @RT(0) @F @F
@END_Algo

@BEG_Dcl
@RT(16)DclTreeContainer
7
@Var @RT(1)b @RT(0) @T @F @DT @RT(4)BOOL @RT(0) @T @T @BASIC 0 @F
@F @F
@T
@BEG_Attrib
3 @RT(0) @RT(0) @RT(0)
@END_Attrib
1 0 @F @F @F @F

@Var @RT(8)activate @RT(0) @T @F @DT @RT(4)DINT @RT(0) @T @T @BASIC 0 @F
@F @F
@T
@BEG_Attrib
3 @RT(0) @RT(0) @RT(0)
@END_Attrib
1 4 @F @F @F @F

@Var @RT(4)name @RT(0) @T @F @DT @RT(11)STRING(255) @RT(0) @T @T @STRING 0 @F @RT(3)255 @F
@F @F
@T
@BEG_Attrib
3 @RT(0) @RT(0) @RT(0)
@END_Attrib
1 0 @F @F @F @F

@Var @RT(1)s @RT(0) @T @T @DERIVED 0 @T @T @DT @RT(11)KSYS_Status @RT(0) @T @T @UNKNOWN 0 @F
@F @F
@T
@BEG_Attrib
3 @RT(0) @RT(0) @RT(0)
@END_Attrib
1 0 @F @F @F @F

@Var @RT(3)cnt @RT(0) @T @F @DT @RT(3)INT @RT(0) @T @T @BASIC 0 @F
@F @F
@T
@BEG_Attrib
3 @RT(0) @RT(0) @RT(0)
@END_Attrib
1 0 @F @F @F @F

@Var @RT(7)cfgFile @RT(0) @T @F @DT @RT(11)STRING(255) @RT(0) @T @T @STRING 0 @F @RT(3)255 @F
@F @F
@T
@BEG_Attrib
3 @RT(0) @RT(0) @RT(0)
@END_Attrib
1 0 @F @F @F @F

@Var @RT(1)i @RT(0) @T @F @DT @RT(4)DINT @RT(0) @T @T @BASIC 0 @F
@F @F
@T
@BEG_Attrib
3 @RT(0) @RT(0) @RT(0)
@END_Attrib
1 4 @F @F @F @F

@END_Dcl

@END_Export

@BEG_Export

@BEG_Algo
@PROCESS_ALGORITHM @RT(6)paInit @STRUCTURED_TEXT
@RT(0) @RT(0) @RT(10)TaskVis(1) @T @F
@END_Algo

@BEG_Dcl
@RT(16)DclTreeContainer
0
@END_Dcl

@END_Export

@BEG_Export

@BEG_Algo
@POSTUPDATE_ALGORITHM @RT(9)pReadDone @STRUCTURED_TEXT
@RT(0) @RT(17)mpiTriggerClient^ @RT(9)PU_Task_3 @F @F
@END_Algo

@BEG_Dcl
@RT(16)DclTreeContainer
0
@END_Dcl

@END_Export

@BEG_Export

@BEG_Algo
@POSTUPDATE_ALGORITHM @RT(9)pActivate @STRUCTURED_TEXT
@RT(0) @RT(32)sv_ProcessDataRecorder.bActivate @RT(9)PU_Task_7 @F @F
@END_Algo

@BEG_Dcl
@RT(16)DclTreeContainer
0
@END_Dcl

@END_Export

@BEG_Export

@BEG_Algo
@POSTUPDATE_ALGORITHM @RT(7)pReload @STRUCTURED_TEXT
@RT(0) @RT(43)sv_ProcessDataRecorder.iReloadConfiguration @RT(7)TaskVis @F @F
@END_Algo

@BEG_Dcl
@RT(16)DclTreeContainer
7
@Var @RT(1)b @RT(0) @T @F @DT @RT(4)BOOL @RT(0) @T @T @BASIC 0 @F
@F @F
@T
@BEG_Attrib
3 @RT(0) @RT(0) @RT(0)
@END_Attrib
1 0 @F @F @F @F

@Var @RT(1)s @RT(0) @T @T @DERIVED 0 @T @T @DT @RT(11)KCAT_Status @RT(0) @T @T @UNKNOWN 0 @F
@F @F
@T
@BEG_Attrib
3 @RT(0) @RT(0) @RT(0)
@END_Attrib
1 0 @F @F @F @F

@Var @RT(10)handleData @RT(0) @T @T @DERIVED 0 @T @T @DT @RT(15)KCAT_HandleData @RT(0) @T @T @UNKNOWN 0 @F
@F @F
@T
@BEG_Attrib
3 @RT(0) @RT(0) @RT(0)
@END_Attrib
1 0 @F @F @F @F

@Var @RT(7)cfgFile @RT(0) @T @F @DT @RT(11)STRING(255) @RT(0) @T @T @STRING 0 @F @RT(3)255 @F
@F @F
@T
@BEG_Attrib
3 @RT(0) @RT(0) @RT(0)
@END_Attrib
1 0 @F @F @F @F

@Var @RT(1)i @RT(0) @T @F @DT @RT(4)DINT @RT(0) @T @T @BASIC 0 @F
@F @F
@T
@BEG_Attrib
3 @RT(0) @RT(0) @RT(0)
@END_Attrib
1 4 @F @F @F @F

@Var @RT(8)workPath @RT(0) @T @F @DT @RT(11)STRING(255) @RT(0) @T @T @STRING 0 @F @RT(3)255 @F
@F @F
@T
@BEG_Attrib
3 @RT(0) @RT(0) @RT(0)
@END_Attrib
1 0 @F @F @F @F

@Var @RT(9)emptyElem @RT(0) @T @T @DERIVED 0 @T @T @DT @RT(11)tsPDRVarRef @RT(0) @T @T @UNKNOWN 0 @F
@F @F
@T
@BEG_Attrib
3 @RT(0) @RT(0) @RT(0)
@END_Attrib
1 15 @F @F @F @F

@END_Dcl

@END_Export

@BEG_Body
@TL(9)
fReadConfigInt := FALSE;
handleData := KCAT_GetHandle(CONCAT(cConfigNode, ".", name));
IF (handleData.Status = KCAT_Status_OK) THEN
    status := KCAT_GetValue(handleData.Handle, value);
    IF (status = KCAT_Status_OK) THEN
        fReadConfigInt := TRUE;
    END_IF;
END_IF;

@END_Body

@@@BEG_Comment@@@
@TL(0)

@@@END_Comment@@@

@BEG_Body
@TL(10)
fReadConfigString := FALSE;
handleData := KCAT_GetHandle(CONCAT(cConfigNode, ".", name));
IF (handleData.Status = KCAT_Status_OK) THEN
    status := KCAT_GetValue(handleData.Handle, value);
    IF (status = KCAT_Status_OK) THEN
        fReadConfigString := TRUE;
    END_IF;
END_IF;

@END_Body

@@@BEG_Comment@@@
@TL(0)

@@@END_Comment@@@

@BEG_Body
@TL(17)
fReadOrAddConfigString := fReadConfigString(name, value);

IF (NOT fReadOrAddConfigString) THEN
        value := default;

        handleData := KCAT_GetHandle(cConfigNode);
        IF (handleData.Status <> KCAT_Status_OK) THEN
            handleData := KCAT_GetRoot();
            handleData := KCAT_AddDir(handleData.Handle, cConfigNode);
        END_IF;
        IF (handleData.Status = KCAT_Status_OK) THEN
            status := KCAT_AddValue(handleData.Handle, name, KCAT_Type_STRING, value);
            fReadOrAddConfigString := status = KCAT_Status_OK;
        END_IF;
END_IF;

@END_Body

@@@BEG_Comment@@@
@TL(0)

@@@END_Comment@@@

@BEG_Body
@TL(14)
IF (mpiTriggerClient^ = 0) THEN
    IF (mReadIdx <> mWriteIdx) THEN
       IF (miMode = 0) THEN
           // sample mode REAL
          sv_ProcessDataRecorder.data := mActProcessData[mReadIdx + 1];
       ELSIF (miMode = 1) THEN
           // sample mode Raw
          sv_ProcessDataRecorder.dataRaw := mActProcessDataRaw[mReadIdx + 1];
       END_IF;
       mReadIdx := (mReadIdx + 1) MOD cPDRMaxLines;
    END_IF;
END_IF;

@END_Body

@@@BEG_Comment@@@
@TL(0)

@@@END_Comment@@@

@BEG_Body
@TL(67)
IF (NOT sv_ProcessDataRecorder.bActivate) THEN
    RETURN;
END_IF;
IF (miMode = 0) THEN
    // sample mode REAL
    FOR i := 1 TO mIdxLastPdrVar DO
        IF (mRecorderConfiguration[i].sampleGroup = iGroupId) THEN
            IF (mRecorderConfiguration[i].prReal <> EMPTY) THEN
                mActProcessData[mWriteIdx+1].yParameter[i] := mRecorderConfiguration[i].prReal^;
            ELSIF (mRecorderConfiguration[i].pdTime <> EMPTY) THEN
                mActProcessData[mWriteIdx+1].yParameter[i] := FTimeToSec(mRecorderConfiguration[i].pdTime^);
            ELSIF (mRecorderConfiguration[i].piDInt <> EMPTY) THEN
                mActProcessData[mWriteIdx+1].yParameter[i] := DINT_TO_REAL(mRecorderConfiguration[i].piDInt^);
            END_IF;
        END_IF;
    END_FOR;
ELSIF (miMode = 1) THEN
    // sample mode RAW
     FOR i := 1 TO mIdxLastPdrVar DO
        IF (mRecorderConfiguration[i].sampleGroup = iGroupId) THEN
            CASE (mRecorderConfiguration[i].nType) OF
                cPDRVarTypeReal:
                    b := CONVERT_LREAL_TO_LWORD(REAL_TO_LREAL(mRecorderConfiguration[i].prReal^), mActProcessDataRaw[mWriteIdx+1].yParameter[i]);

                cPDRVarTypeTime:
                    mActProcessDataRaw[mWriteIdx+1].yParameter[i] := LINT_TO_LWORD(TIME_TO_LINT(mRecorderConfiguration[i].pdTime^));

                cPDRVarTypeDInt:
                    mActProcessDataRaw[mWriteIdx+1].yParameter[i] := LINT_TO_LWORD(DINT_TO_LINT(mRecorderConfiguration[i].piDInt^));

                cPDRVarTypeLReal:
                    b := CONVERT_LREAL_TO_LWORD(mRecorderConfiguration[i].prLReal^, mActProcessDataRaw[mWriteIdx+1].yParameter[i]);

                cPDRVarTypeBool:
                    mActProcessDataRaw[mWriteIdx+1].yParameter[i] := LINT_TO_LWORD(BOOL_TO_LINT(mRecorderConfiguration[i].pbBool^));

                cPDRVarTypeDT:
                    mActProcessDataRaw[mWriteIdx+1].yParameter[i] := LINT_TO_LWORD(DATE_TO_LINT(DT_TO_DATE(mRecorderConfiguration[i].pdDT^))+TIME_TO_LINT(TOD_TO_TIME(DT_TO_TOD(mRecorderConfiguration[i].pdDT^))));

                cPDRVarTypeSInt:
                    mActProcessDataRaw[mWriteIdx+1].yParameter[i] := LINT_TO_LWORD(SINT_TO_LINT(mRecorderConfiguration[i].piSInt^));

                cPDRVarTypeInt:
                    mActProcessDataRaw[mWriteIdx+1].yParameter[i] := LINT_TO_LWORD(INT_TO_LINT(mRecorderConfiguration[i].piInt^));

                cPDRVarTypeLInt:
                    mActProcessDataRaw[mWriteIdx+1].yParameter[i] := LINT_TO_LWORD(mRecorderConfiguration[i].piLInt^);

                cPDRVarTypeUSInt:
                    mActProcessDataRaw[mWriteIdx+1].yParameter[i] := USINT_TO_LWORD(mRecorderConfiguration[i].piUSInt^);

                cPDRVarTypeUInt:
                    mActProcessDataRaw[mWriteIdx+1].yParameter[i] := UINT_TO_LWORD(mRecorderConfiguration[i].piUInt^);

                cPDRVarTypeUDInt:
                    mActProcessDataRaw[mWriteIdx+1].yParameter[i] := UDINT_TO_LWORD(mRecorderConfiguration[i].piUDInt^);

                cPDRVarTypeULInt:
                    mActProcessDataRaw[mWriteIdx+1].yParameter[i] := ULINT_TO_LWORD(mRecorderConfiguration[i].piULInt^);

             END_CASE;
        END_IF;
    END_FOR;
END_IF;

@END_Body

@@@BEG_Comment@@@
@TL(0)

@@@END_Comment@@@

@BEG_Body
@TL(33)
(**************************************** WARNING ********************************************
 *** The KEBA Kemro K2 System including software is not intended for safety control tasks! ***
 ***                       For further information see Comment tab!                        ***
 *********************************************************************************************)

ts := GET_RUNTIME();
aDoSample(0);
fbRtc();

IF (miMode = 0) THEN
    // sample mode REAL
    mActProcessData[mWriteIdx+1].iTrigger := mpiTriggerPU^;
    mActProcessData[mWriteIdx+1].dTimeStamp := fbRtc.CDT;
    mWriteIdx := (mWriteIdx + 1) MOD cPDRMaxLines;
    mActProcessData[mWriteIdx + 1].yParameter := emptyProcessData;
    mActProcessData[mWriteIdx + 1].iTrigger := 0;
ELSIF (miMode = 1) THEN
    // sample mode RAW
    mActProcessDataRaw[mWriteIdx+1].iTrigger := mpiTriggerPU^;
    mActProcessDataRaw[mWriteIdx+1].dTimeStamp := fbRtc.CDT;
    mWriteIdx := (mWriteIdx + 1) MOD cPDRMaxLines;
    mActProcessDataRaw[mWriteIdx + 1].yParameter := emptyProcessDataRaw;
    mActProcessDataRaw[mWriteIdx + 1].iTrigger := 0;
END_IF;

IF (mWriteIdx = mReadIdx) THEN
    mReadIdx := (mReadIdx + 1) MOD cPDRMaxLines;
END_IF;

aSignalRead();

t := GET_RUNTIME() - ts;

@END_Body

@@@BEG_Comment@@@
@TL(11)
@h    ! WARNING !
@h    The Kemro K2 system (including software) only meets category B according to EN 954-1,
@h    thus it is not intended for usage in safety-relevant control applications in the field
@h    of personal safety (e.g. emergency stop).
@h    To implement potentially necessary safety-relevant control tasks, always use additional
@h    external safety devices that are intended for the particular purpose, and meet the necessary
@h    functional safety.
@h    For further information see EN 954-1 (EN ISO 13849-1) and/or the K2-x00 user manual, chapter
@h    "CE conformity, directives and standards".

@@@END_Comment@@@

@BEG_Body
@TL(15)
(**************************************** WARNING ********************************************
 *** The KEBA Kemro K2 System including software is not intended for safety control tasks! ***
 ***                       For further information see Comment tab!                        ***
 *********************************************************************************************)

IF ((evMovementStateData.DeviceId.CompId = cCompInjection)
   AND (evMovementStateData.DeviceId.IndexId = 1)
   AND (evMovementStateData.MoveId   = cMoveInject)
   AND (evMovementStateData.MoveDir  = cMoveFwd)
   AND (evMovementStateData.State  = nActive)) THEN

    // copy data at inject time
    aDoSample(16);
END_IF;

@END_Body

@@@BEG_Comment@@@
@TL(11)
@h    ! WARNING !
@h    The Kemro K2 system (including software) only meets category B according to EN 954-1,
@h    thus it is not intended for usage in safety-relevant control applications in the field
@h    of personal safety (e.g. emergency stop).
@h    To implement potentially necessary safety-relevant control tasks, always use additional
@h    external safety devices that are intended for the particular purpose, and meet the necessary
@h    functional safety.
@h    For further information see EN 954-1 (EN ISO 13849-1) and/or the K2-x00 user manual, chapter
@h    "CE conformity, directives and standards".

collects processdata: sample values at inject
@@@END_Comment@@@

@BEG_Body
@TL(130)
b := fReadOrAddConfigString(cConfigNodeCfgFile, cfgFile, 'workspace/data/pdr.cfg');

miMode := 0;
b := fReadConfigInt("Mode", miMode);
b := fReadConfigInt("Activate", activate);

IF (fReadConfigString("Trigger", name)) THEN
   mpiTrigger := GET_SYNC_REFTO(name, T#0s, s);
END_IF;

IF (mpiTrigger = EMPTY) THEN
    mpiTrigger := @sv_iShotCounterAct;
END_IF;

FOR i := 1 TO cPDRMaxVars DO
   mRecorderConfiguration[i].nType := cPDRVarTypeNone;
   IF (fReadConfigString(CONCAT("Var:", DINT_TO_STRING(i), ".Name"), name)) THEN

       /////////   R E A L   /////////
       IF (mRecorderConfiguration[i].nType = cPDRVarTypeNone) THEN
          mRecorderConfiguration[i].prReal := GET_SYNC_REFTO(name, T#0s, s);
          IF (s = KSYS_Status_OK) THEN
             mRecorderConfiguration[i].nType := cPDRVarTypeReal;
          END_IF;
       END_IF;
       /////////   T I M E   /////////
       IF (mRecorderConfiguration[i].nType = cPDRVarTypeNone) THEN
          mRecorderConfiguration[i].pdTime := GET_SYNC_REFTO(name, T#0s, s);
          IF (s = KSYS_Status_OK) THEN
             mRecorderConfiguration[i].nType := cPDRVarTypeTime;
          END_IF;
       END_IF;
       /////////   D I N T   /////////
       IF (mRecorderConfiguration[i].nType = cPDRVarTypeNone) THEN
          mRecorderConfiguration[i].piDInt := GET_SYNC_REFTO(name, T#0s, s);
          IF (s = KSYS_Status_OK) THEN
             mRecorderConfiguration[i].nType := cPDRVarTypeDInt;
          END_IF;
       END_IF;

       IF (miMode > 0) THEN
            /////////   L R E A L   /////////
            IF (mRecorderConfiguration[i].nType = cPDRVarTypeNone) THEN
                mRecorderConfiguration[i].prLReal := GET_SYNC_REFTO(name, T#0s, s);
                IF (s = KSYS_Status_OK) THEN
                    mRecorderConfiguration[i].nType := cPDRVarTypeLReal;
                END_IF;
            END_IF;
            /////////   B O O L   /////////
            IF (mRecorderConfiguration[i].nType = cPDRVarTypeNone) THEN
                mRecorderConfiguration[i].pbBool := GET_SYNC_REFTO(name, T#0s, s);
                IF (s = KSYS_Status_OK) THEN
                    mRecorderConfiguration[i].nType := cPDRVarTypeBool;
                END_IF;
            END_IF;
            /////////   D A T E  &  T I M E   /////////
            IF (mRecorderConfiguration[i].nType = cPDRVarTypeNone) THEN
                mRecorderConfiguration[i].pdDT := GET_SYNC_REFTO(name, T#0s, s);
                IF (s = KSYS_Status_OK) THEN
                    mRecorderConfiguration[i].nType := cPDRVarTypeDT;
                END_IF;
            END_IF;
            /////////   S I N T   /////////
            IF (mRecorderConfiguration[i].nType = cPDRVarTypeNone) THEN
                mRecorderConfiguration[i].piSInt := GET_SYNC_REFTO(name, T#0s, s);
                IF (s = KSYS_Status_OK) THEN
                    mRecorderConfiguration[i].nType := cPDRVarTypeSInt;
                END_IF;
            END_IF;
            /////////   I N T   /////////
            IF (mRecorderConfiguration[i].nType = cPDRVarTypeNone) THEN
                mRecorderConfiguration[i].piInt := GET_SYNC_REFTO(name, T#0s, s);
                IF (s = KSYS_Status_OK) THEN
                    mRecorderConfiguration[i].nType := cPDRVarTypeInt;
                END_IF;
            END_IF;
            /////////   L I N T   /////////
            IF (mRecorderConfiguration[i].nType = cPDRVarTypeNone) THEN
                mRecorderConfiguration[i].piLInt := GET_SYNC_REFTO(name, T#0s, s);
                IF (s = KSYS_Status_OK) THEN
                    mRecorderConfiguration[i].nType := cPDRVarTypeLInt;
                END_IF;
            END_IF;
            /////////   U S I N T   /////////
            IF (mRecorderConfiguration[i].nType = cPDRVarTypeNone) THEN
                mRecorderConfiguration[i].piUSInt := GET_SYNC_REFTO(name, T#0s, s);
                IF (s = KSYS_Status_OK) THEN
                    mRecorderConfiguration[i].nType := cPDRVarTypeUSInt;
                END_IF;
            END_IF;
                /////////   U I N T   /////////
            IF (mRecorderConfiguration[i].nType = cPDRVarTypeNone) THEN
                mRecorderConfiguration[i].piUInt := GET_SYNC_REFTO(name, T#0s, s);
                IF (s = KSYS_Status_OK) THEN
                    mRecorderConfiguration[i].nType := cPDRVarTypeUInt;
                END_IF;
            END_IF;
            /////////   U D I N T   /////////
            IF (mRecorderConfiguration[i].nType = cPDRVarTypeNone) THEN
                mRecorderConfiguration[i].piUDInt := GET_SYNC_REFTO(name, T#0s, s);
                IF (s = KSYS_Status_OK) THEN
                    mRecorderConfiguration[i].nType := cPDRVarTypeUDInt;
                END_IF;
            END_IF;
            /////////   U L I N T   /////////
            IF (mRecorderConfiguration[i].nType = cPDRVarTypeNone) THEN
                mRecorderConfiguration[i].piULInt := GET_SYNC_REFTO(name, T#0s, s);
                IF (s = KSYS_Status_OK) THEN
                    mRecorderConfiguration[i].nType := cPDRVarTypeULInt;
                END_IF;
            END_IF;
       END_IF;

       // Type found ... save last used index in configuration
       IF (mRecorderConfiguration[i].nType <> cPDRVarTypeNone) THEN
          mIdxLastPdrVar := i;
       END_IF;

       cnt := cnt + 1;
       b := fReadConfigInt(CONCAT("Var:", DINT_TO_STRING(i), ".SampleGroup"), mRecorderConfiguration[i].sampleGroup);
   END_IF;
   sv_ProcessDataRecorder.yActiveVariables[i] := mRecorderConfiguration[i].nType;
END_FOR;

IF (activate <> 0) THEN
    sv_ProcessDataRecorder.bActivate := TRUE;
END_IF;

@END_Body

@@@BEG_Comment@@@
@TL(0)

@@@END_Comment@@@

@BEG_Body
@TL(4)
STOP_PROCESS_ALGORITHM();

aInit();

@END_Body

@@@BEG_Comment@@@
@TL(0)

@@@END_Comment@@@

@BEG_Body
@TL(2)
aSignalRead();

@END_Body

@@@BEG_Comment@@@
@TL(0)

@@@END_Comment@@@

@BEG_Body
@TL(18)
IF (sv_ProcessDataRecorder.bActivate) THEN
   mpiTriggerPU := mpiTrigger;
   mevMovementState := evMovementState;
   IF (miMode = 0) THEN
       // sample mode real
       mpiTriggerClient := @sv_ProcessDataRecorder.data.iTrigger;
   ELSIF (miMode = 1) THEN
       // sample mode raw
       mpiTriggerClient := @sv_ProcessDataRecorder.dataRaw.iTrigger;
   END_IF;
ELSE
   mpiTriggerPU := EMPTY;
   mevMovementState := EMPTY;
   mpiTriggerClient := EMPTY;
END_IF;

@END_Body

@@@BEG_Comment@@@
@TL(0)

@@@END_Comment@@@

@BEG_Body
@TL(31)
IF (sv_ProcessDataRecorder.iReloadConfiguration MOD 2 = 1) THEN
    sv_ProcessDataRecorder.bActivate := FALSE;

    cfgFile := "";
    b := fReadConfigString(cConfigNodeCfgFile, cfgFile);
    handleData := KCAT_GetHandle(cConfigNode);
    IF (handleData.Status = KCAT_Status_OK) THEN
        s := KCAT_RemoveDir(handleData.Handle);
    END_IF;

    workPath := FGetCatConfigValueString("System.workPath", "/");

    FOR i := 1 TO cPDRMaxVars DO
        mRecorderConfiguration[i] := emptyElem;
    END_FOR;

    mWriteIdx := 0;
    mReadIdx := 0;

    s := KCAT_Load(CONCAT(workPath, "/", cfgFile));

    aInit();

    IF (LEN(cfgFile) > 0) THEN
      b := fReadOrAddConfigString(cConfigNodeCfgFile, cfgFile, cfgFile);
    END_IF;

    sv_ProcessDataRecorder.iReloadConfiguration := sv_ProcessDataRecorder.iReloadConfiguration + 1;
END_IF;

@END_Body

@@@BEG_Comment@@@
@TL(0)

@@@END_Comment@@@
@END_Body

@END_Contents

(* ---- FCreateHostComVersion.pu ---- *)
(*
@h    ! WARNING !
@h    The Kemro K2 system (including software) only meets category B according to EN 954-1,
@h    thus it is not intended for usage in safety-relevant control applications in the field
@h    of personal safety (e.g. emergency stop).
@h    To implement potentially necessary safety-relevant control tasks, always use additional
@h    external safety devices that are intended for the particular purpose, and meet the necessary
@h    functional safety.
@h    For further information see EN 954-1 (EN ISO 13849-1) and/or the K2-x00 user manual, chapter
@h    "CE conformity, directives and standards".

this file is automatically created by clearcase makebaseline
and contains versioninformation of component
*)

IMPORT_OVER_LISTFILE
 FWriteComponentVersion

END_IMPORT

FUNCTION FCreateHostComVersion : BOOL #DUMMY_EDIT_BLOCK

VAR CONSTANT
 sComponentName : STRING(255) := 'ApplMoldMachineOptions.HostCommunication';
 iComponentNumber : DINT := 6597;
 sVersionString : STRING(255) := '01.56';
 iVersionMajor : DINT := 1;
 iVersionMinor : DINT := 56;
END_VAR
#BEGIN_EDIT_BLOCK
(**************************************** WARNING ********************************************
 *** The KEBA Kemro K2 System including software is not intended for safety control tasks! ***
 ***                       For further information see Comment tab!                        ***
 *********************************************************************************************)

FCreateHostComVersion := FWriteComponentVersion(
        sComponentName,
        iComponentNumber,
        sVersionString,
        iVersionMajor,
        iVersionMinor
);

;#END_EDIT_BLOCK END_FUNCTION

#END_OF_IEC_PART

@Puma @IecEditor 6 68 @Pou 25
@@@BEG_Comment@@@
@h    ! WARNING !
@h    The Kemro K2 system (including software) only meets category B according to EN 954-1,
@h    thus it is not intended for usage in safety-relevant control applications in the field
@h    of personal safety (e.g. emergency stop).
@h    To implement potentially necessary safety-relevant control tasks, always use additional
@h    external safety devices that are intended for the particular purpose, and meet the necessary
@h    functional safety.
@h    For further information see EN 954-1 (EN ISO 13849-1) and/or the K2-x00 user manual, chapter
@h    "CE conformity, directives and standards".

this file is automatically created by clearcase makebaseline
and contains versioninformation of component
@@@END_Comment@@@

@BEG_Contents

@BEG_Func
@RT(17)FuncTreeContainer
1
@Var @RT(22)FWriteComponentVersion @RT(0) @T @F @DT @RT(0) @RT(0) @T @T @UNKNOWN 0 @F
@F @F
@T
@BEG_Attrib
0 @RT(0) @RT(0)
@END_Attrib
1 1 @F @F @F @F

@END_Func

@BEG_Const
@RT(18)ConstTreeContainer
0
@END_Const

@BEG_Export

@BEG_Kind
@FUNCTION @RT(21)FCreateHostComVersion @STRUCTURED_TEXT
@RT(4)BOOL @RT(0) @RT(0)
@END_Kind

@BEG_Dcl
@RT(16)DclTreeContainer
5
@Var @RT(14)sComponentName @RT(0) @T @F @DT @RT(11)STRING(255) @RT(0) @T @T @STRING 0 @F @RT(3)255 @F
@F @F
@T
@BEG_Attrib
3 @RT(42)'ApplMoldMachineOptions.HostCommunication' @RT(0) @RT(0)
@END_Attrib
1 15 @F @F @F @F

@Var @RT(16)iComponentNumber @RT(0) @T @F @DT @RT(4)DINT @RT(0) @T @T @BASIC 0 @F
@F @F
@T
@BEG_Attrib
3 @RT(4)6597 @RT(0) @RT(0)
@END_Attrib
1 15 @F @F @F @F

@Var @RT(14)sVersionString @RT(0) @T @F @DT @RT(11)STRING(255) @RT(0) @T @T @STRING 0 @F @RT(3)255 @F
@F @F
@T
@BEG_Attrib
3 @RT(7)'01.56' @RT(0) @RT(0)
@END_Attrib
1 15 @F @F @F @F

@Var @RT(13)iVersionMajor @RT(0) @T @F @DT @RT(4)DINT @RT(0) @T @T @BASIC 0 @F
@F @F
@T
@BEG_Attrib
3 @RT(1)1 @RT(0) @RT(0)
@END_Attrib
1 15 @F @F @F @F

@Var @RT(13)iVersionMinor @RT(0) @T @F @DT @RT(4)DINT @RT(0) @T @T @BASIC 0 @F
@F @F
@T
@BEG_Attrib
3 @RT(2)56 @RT(0) @RT(0)
@END_Attrib
1 15 @F @F @F @F

@END_Dcl

@END_Export

@BEG_Body
@TL(13)
(**************************************** WARNING ********************************************
 *** The KEBA Kemro K2 System including software is not intended for safety control tasks! ***
 ***                       For further information see Comment tab!                        ***
 *********************************************************************************************)

FCreateHostComVersion := FWriteComponentVersion(
        sComponentName,
        iComponentNumber,
        sVersionString,
        iVersionMajor,
        iVersionMinor
);

@END_Body

@END_Contents

(* ---- FHostTypeToString.pu ---- *)
IMPORT_OVER_LISTFILE
 cHostTypeNone
, cHostTypeOPCGeneric
, cHostTypeOPC_EM63

END_IMPORT

FUNCTION FHostTypeToString : STRING(32) #DUMMY_EDIT_BLOCK

VAR_INPUT
 iHostType : DINT;
END_VAR
#BEGIN_EDIT_BLOCK
CASE (iHostType) OF
   cHostTypeOPCGeneric:
      FHostTypeToString := "OPC Generic";

   cHostTypeOPC_EM63:
      FHostTypeToString := "EM63 over OPC";

   cHostTypeOPCUA_EM77:
      FHostTypeToString := "EM77 over OPCUA";

ELSE
   FHostTypeToString := "invalid id";
END_CASE;

;#END_EDIT_BLOCK END_FUNCTION

#END_OF_IEC_PART

@Puma @IecEditor 6 159 @Pou 25
@@@BEG_Comment@@@

@@@END_Comment@@@

@BEG_Contents

@BEG_Func
@RT(17)FuncTreeContainer
0
@END_Func

@BEG_Const
@RT(18)ConstTreeContainer
3
@Var @RT(13)cHostTypeNone @RT(0) @T @F @DT @RT(4)DINT @RT(0) @T @T @BASIC 0 @F
@F @F
@T
@BEG_Attrib
0 @RT(1)0 @RT(0)
@END_Attrib
1 1 @F @F @F @F

@Var @RT(19)cHostTypeOPCGeneric @RT(0) @T @F @DT @RT(4)DINT @RT(0) @T @T @BASIC 0 @F
@F @F
@T
@BEG_Attrib
0 @RT(1)1 @RT(0)
@END_Attrib
1 1 @F @F @F @F

@Var @RT(17)cHostTypeOPC_EM63 @RT(0) @T @F @DT @RT(4)DINT @RT(0) @T @T @BASIC 0 @F
@F @F
@T
@BEG_Attrib
0 @RT(1)2 @RT(0)
@END_Attrib
1 1 @F @F @F @F

@END_Const

@BEG_Export

@BEG_Kind
@FUNCTION @RT(17)FHostTypeToString @STRUCTURED_TEXT
@RT(10)STRING(32) @RT(0) @RT(0)
@END_Kind

@BEG_Dcl
@RT(16)DclTreeContainer
1
@Var @RT(9)iHostType @RT(0) @T @F @DT @RT(4)DINT @RT(0) @T @T @BASIC 0 @F
@F @F
@T
@BEG_Attrib
3 @RT(0) @RT(0) @RT(0)
@END_Attrib
1 1 @F @F @F @F

@END_Dcl

@END_Export

@BEG_Body
@TL(14)
CASE (iHostType) OF
   cHostTypeOPCGeneric:
      FHostTypeToString := "OPC Generic";

   cHostTypeOPC_EM63:
      FHostTypeToString := "EM63 over OPC";

   cHostTypeOPCUA_EM77:
      FHostTypeToString := "EM77 over OPCUA";

ELSE
   FHostTypeToString := "invalid id";
END_CASE;

@END_Body

@END_Contents
